(* CODESYS project Base_Elements.library
   Company: Vistaprint
   Title: Base_Elements
   Description: 0.0.1.22 - FB_UMC Always SingleAnswer 
      0.0.1.21 - Added GHT (10Digit Key compatible Hash)
      0.0.1.20 - Added newest BasePLC, addapted main component controll
      0.0.1.19 - Added newest EtherCat Library version
      0.0.1.18 - FB_BCC RP-208 - Implement sensor signal input for triggering a barcode scan
      0.0.1.17 - DRV Main Switch added
      0.0.1.16 - Added the Generic DataChannels
      0.0.1.15 - Added new BaseConcept Lib V0.3.4.8
      0.0.1.14 - Added new BaseConcept Lib
      0.0.1.13 - Changes in timeout handling BaseCtrlModule. Inserted new parameter  udiTimeoutStarting_ms. TO handling can now switched off with value 0.
      0.0.1.12 - Added new base_class
      0.0.1.11 - Bugfix in UMC
      0.0.1.10 - SGT added
      0.0.1.9 - Newest Base_PLC added 0.3.4.5
      0.0.1.8 - Integrate ECD (EtherCAT Diagnostic)
      0.0.1.7 - More RFW Error information
      0.0.1.5 - Added new controller FB_VLV
      0.0.1.4 - Fix for the BCD, BCC controller to support also messages without diagnostics
      0.0.1.2 - Simulation UMC; FB_CtrlModule added
      0.0.1.1 - Newest Base_PLC added 0.3.4.2
      0.0.1.0 - Newest Base_PLC added 0.3.4.0
      - FB_RFW Bug fix write single data
      0.0.0.26 - FB_ACL Enter ADS route string automatically during state PONBusy.
      0.0.0.25 - DLL FUB added
      0.0.0.24 - EOFFbusy Fix in FB_UMC
      0.0.0.23 - New ADS Client FUB (ACL) added
      	Sample added in MiddleTask
      0.0.0.22 - UMC simulation added, Refactoring
      0.0.0.21 - UMC - Add EMO State, Refactoring
      0.0.0.20 - New version of BCD and BCC
      0.0.0.19 - Back to BasePLC Lib. V3.3.5 beacuase of PageFaults
      0.0.0.18 - RFW integrated from Promp
      0.0.0.17 - DRV added
      0.0.0.16 - Newest Base_PLC added 0.3.3.7
      0.0.0.15 - Basic versions of Barcode driver and controller added
      0.0.0.11 - Newest Base_PLC added
      0.0.0.10 - Newest Base_PLC added
      0.0.0.9 - Add cylinder Level0, Update to Base PLC 0.3.3.2
      0.0.0.8 - Update to Base PLC 0.3.3.0
      0.0.0.7 - Updated to newest tc2_utilities
      0.0.0.6 - Added the PRS controller
      0.0.0.5 - Added the UMC and VPC controller
   Author: DSC - KVO
   Version: 0.0.1.22

Project tree, tasks and I/O mapping:
  libraries: Base_PLC, 0.3.4.9 (Vistaprint); Tc2_EtherCAT, 3.3.3.0 (Beckhoff Automation GmbH); Tc2_SerialCom, 3.3.2.0 (Beckhoff Automation GmbH); Tc2_Standard, 3.3.0.0 (Beckhoff Automation GmbH); Tc2_System, 3.3.5.0 (Beckhoff Automation GmbH); Tc2_TcpIp, 3.3.2.0 (Beckhoff Automation GmbH); Tc2_Utilities, 3.3.7.0 (Beckhoff Automation GmbH); Tc3_Interfaces, 3.3.0.0 (Beckhoff Automation GmbH); Tc3_MemMan, 3.3.1.0 (Beckhoff Automation GmbH); Tc3_Module, 3.3.5.0 (Beckhoff Automation GmbH)
  POUs/
    Controller/
      Driver/
        ACL (ADS client for data exchange)/
          global variables ACL_Const
          global variables ADS_IndexGroup
          data type E_ADS_AccessType
          function block FB_ACL [ST]: AddConnection, Always, FB_init, getCmdState, getCtrlSIf, GetNextAccessType, NetIDtoAddress, sta_ERROR, sta_OFF, sta_PON, sta_PONBusy, sta_RUN, sta_RUNBusy, StateMachine
          data type T_ADS_ConnectionData
          data type T_Ctrl_SIf_ACL
          data type T_Ctrl_SIf_ACL_Cur
          data type T_Ctrl_SIf_ACL_Par
        BCD (Bar code driver)/
          global variables BCD_CmdState
          function block FB_BCD [ST]: CheckSensorError, CtrlInit, CycleEndDuty, CycleStartDuty, FB_init, getCmdState, getSIf, HandleRxData, HandleTxData, PrepareBarCodeData, PrepareReadMsg, PrepareSendMsg, sta_CloseSocketBusy, sta_ComTestBusy, sta_ConnectSocketBusy, sta_Error, sta_ReadCodeBusy, sta_SocketClosed, sta_WaitForJob, StateMachine
          function FC_StrComp [ST]
          data type T_BCD
          data type T_BCD_Cfg
          data type T_BCD_Data
          data type T_BCD_DeviceInfo
          data type T_BCD_Error
          data type T_BCD_OperatingData
          data type T_BCD_Par
          data type T_BCD_ServiceInfo
          data type T_BCD_StateMachine
          data type T_BCD_Status
        PRS [Present Sensor]/
          data type E_ALM_PRS
          function block FB_PRS [ST]: Always, CtrlSIf, FB_init, getCmdState, getCtrlSIf, IoInBridge, IoOutBridge, sta_ABSENT, sta_ABSENTBusy, sta_PON, sta_PRESENT, sta_PRESENTBusy, StateMachine
          global variables PRS_CmdState
          data type T_Ctrl_SIf_PRS
          data type T_Ctrl_SIf_PRS_Cfg
          data type T_Ctrl_SIf_PRS_Cur
          data type T_Ctrl_SIf_PRS_Ilk
          data type T_Ctrl_SIf_PRS_In
          data type T_Ctrl_SIf_PRS_Out
          data type T_Ctrl_SIf_PRS_Par
        RFD (RFID Driver)/
          data type E_Typ_Baudrate
          data type E_Typ_Ftim
          function block FB_Com_3964R [ST]
          function block FB_ExCom [ST]
          function FB_HEXSTRING_TO_ULINT [ST]
          function block FB_RFD [ST]: CtrlInit, CycleEndDuty, CycleStartDuty, FB_init, getCmdState, getSIf, sta_CheckBusy, sta_Error, sta_MDSBusy, sta_Off, sta_OffBusy, sta_PowerOnBusy, sta_ReadBusy, sta_SLGBusy, sta_TagInitBusy, sta_WaitForJob, sta_WriteBusy, StateMachine, StateMachine_Service
          function block FB_RFR [ST]: CtrlInit, CycleEndDuty, CycleStartDuty, FB_init, getCmdState, getSIf, sta_Error, sta_PowerOnBusy, sta_WaitForJob, StateMachine, StateMachine_Service
          global variables RFD_Cmd
          global variables RFD_Constants
          data type T_RFD
          data type T_RFD_Cfg
          data type T_RFD_Cur
          data type T_RFD_Error
          data type T_RFD_MDS_Diagnose
          data type T_RFD_MDS_State
          data type T_RFD_SLG_Diagnose
          data type T_RFD_SLG_State
          data type T_RFD_StateMachine
          data type T_RFD_Status
          data type T_StateWord
      Lvl0/
        BCC (Barcode controller)/
          global variables BCC_CmdState
          function block FB_BCC [ST]: Always, FB_init, getCmdState, getCtrlSIf, IoInBridge, IoOutBridge, sta_ERROR, sta_OFF, sta_OFFBusy, sta_PON, sta_PONBusy, sta_READ, sta_READBusy, StateMachine
          data type T_BCC_Data
          data type T_Ctrl_SIf_BCC
          data type T_Ctrl_SIf_BCC_Cfg
          data type T_Ctrl_SIf_BCC_Cur
          data type T_Ctrl_SIf_BCC_In
          data type T_Ctrl_SIf_BCC_Out
          data type T_Ctrl_SIf_BCC_Par
        CYL (Cylinder)/
          global variables CYL_CmdState
          data type E_ALM_CYL
          data type E_Typ_CYL
          function block FB_CYL [ST]: Always, FB_init, getCmdState, getCtrlSIf, IoInBridge, IoOutBridge, sta_ERROR, sta_ERRORQuit, sta_EXTEND, sta_EXTENDBusy, sta_OFF, sta_OFFBusy, sta_RETRACT, sta_RETRACTBusy, sta_STOP, sta_STOPBusy, StateMachine
          data type T_Ctrl_SIf_CYL
          data type T_Ctrl_SIf_CYL_Cfg
          data type T_Ctrl_SIf_CYL_Cur
          data type T_Ctrl_SIf_CYL_Ilk
          data type T_Ctrl_SIf_CYL_In
          data type T_Ctrl_SIf_CYL_Out
          data type T_Ctrl_SIf_CYL_Par
        DRV (Drive)/
          global variables Const_DRV
          data type E_Typ_DRV
          function block FB_DRV [ST]: Always, FB_init, getCtrlSIf, IoInBridge, IoOutBridge, SetSpeed, sta_ERROR, sta_OFF, sta_OFFBusy, sta_PON, sta_RUN, sta_RUNBusy, StateMachine
          data type T_Ctrl_SIf_DRV
          data type T_Ctrl_SIf_DRV_Cfg
          data type T_Ctrl_SIf_DRV_Cur
          data type T_Ctrl_SIf_DRV_In
          data type T_Ctrl_SIf_DRV_Out
          data type T_Ctrl_SIf_DRV_Par
        ECD (EtherCAT Diagnostic)/
          data type E_ALM_ECD
          global variables ECD_Const
          function block FB_ECD [ST]: Always, FB_init, getCmdState, getCtrlSIf, sta_ERROR, sta_ERRORQuit, sta_OFF, sta_PON, sta_PONBusy, sta_RUN, sta_RUNBusy, StateMachine
          data type T_Ctrl_SIf_ECD
          data type T_Ctrl_SIf_ECD_Cfg
          data type T_Ctrl_SIf_ECD_Cur
          data type T_Ctrl_SIf_ECD_Par
          data type T_ECD_SlaveData
        RFW (RFID Reader-Writer)/
          data type E_Typ_RFW
          function block FB_DtChnToLine_NewRFID [ST]: Creat
          function block FB_RFW [ST]: Always, FB_init, getCmdState, getCtrlSIf, IoInBridge, IoOutBridge, sta_ERROR, sta_OFF, sta_OFFBusy, sta_ON, sta_ONbusy, sta_PON, sta_PONBusy, sta_READ, sta_READBusy, sta_RUN, sta_RUNbusy, sta_WRITE, sta_WRITEBusy, StateMachine
          function FB_ULINT_TO_HEXSTRING [ST]
          global variables RFID_Data
          global variables RFW_CmdState
          data type T_Ctrl_SIf_RFW
          data type T_Ctrl_SIf_RFW_Cfg
          data type T_Ctrl_SIf_RFW_Cur
          data type T_Ctrl_SIf_RFW_DtChnToLine
          data type T_Ctrl_SIf_RFW_In
          data type T_Ctrl_SIf_RFW_Out
          data type T_Ctrl_SIf_RFW_Par
          data type T_NewRFID_DtChn
          data type T_RFW
        SGT (Signal Tower)/
          data type E_ALM_SGT
          function block FB_SGT [ST]: Always, FB_init, getCmdState, getCtrlSIf, IoOutBridge, setBeepOutput, setLampOutput, sta_OFF, sta_OFFBusy, sta_PON, sta_PONBusy, sta_RUN, sta_RUNBusy, StateMachine
          data type T_Ctrl_SIf_SGT
          data type T_Ctrl_SIf_SGT_Cfg
          data type T_Ctrl_SIf_SGT_Out
          data type T_Ctrl_SIf_SGT_Par
        UMC [Universal Motor Controller]/
          data type E_ALM_UMC
          data type E_CFG_UMC
          data type E_TURN_DIRECTION
          data type E_UMC_MOTOR_STATUS
          function block FB_UMC [ST]: Always, cmd_MotorOff, cmd_MotorOn, cmd_MotorReset, cmd_MotorStop, CtrlInit, CtrlSIf, CycleEndDuty, CycleStartDuty, FB_init, getCmdState, getCtrlSIf, GetMotorStatus, GetSpeedValue, IoInBridge, IoOutBridge, sta_EOFF, sta_EOFFbusy, sta_ERROR, sta_ERRORQuit, sta_OFF, sta_OFFBusy, sta_PON, sta_RESETMOTORERROR, sta_RUN, sta_RUNBusy, sta_SETOPERATIONMODE, sta_STOP, sta_STOPBusy, StateMachine
          data type T_Ctrl_SIf_UMC
          data type T_Ctrl_SIf_UMC_Cfg
          data type T_Ctrl_SIf_UMC_Cur
          data type T_Ctrl_SIf_UMC_Ilk
          data type T_Ctrl_SIf_UMC_In
          data type T_Ctrl_SIf_UMC_Out
          data type T_Ctrl_SIf_UMC_Par
          data type T_UMC_Lenze_Control
          data type T_UMC_Lenze_Status
          data type U_UMC_Lenze_Control
          data type U_UMC_Lenze_Status
          global variables UMC_CmdState
        VLV (Valve controller)/
          data type E_ALM_VLV
          data type E_Typ_VLV
          function block FB_VLV [ST]: Always, FB_init, getCmdState, getCtrlSIf, IoInBridge, IoOutBridge, sta_CLOSE, sta_CLOSEBusy, sta_ERROR, sta_ERRORQuit, sta_OFF, sta_OFFBusy, sta_OPEN, sta_OPENBusy, StateMachine
          data type T_Ctrl_SIf_VLV
          data type T_Ctrl_SIf_VLV_Cfg
          data type T_Ctrl_SIf_VLV_Cur
          data type T_Ctrl_SIf_VLV_Ilk
          data type T_Ctrl_SIf_VLV_In
          data type T_Ctrl_SIf_VLV_Out
          data type T_Ctrl_SIf_VLV_Par
          global variables VLV_CmdState
        VPC [Vacuum Pump Controller]/
          data type E_ALM_VPC
          data type E_CFG_VPC
          function block FB_VPC [ST]: Always, FB_init, getCmdState, getCtrlSIf, IoInBridge, IoOutBridge, sta_ERROR, sta_ERRORQuit, sta_OFF, sta_OFFBusy, sta_PON, sta_RUN, sta_RUNBusy, sta_StabilizeVacuum, StateMachine
          data type T_Ctrl_SIf_VPC
          data type T_Ctrl_SIf_VPC_Cfg
          data type T_Ctrl_SIf_VPC_Cur
          data type T_Ctrl_SIf_VPC_Ilk
          data type T_Ctrl_SIf_VPC_In
          data type T_Ctrl_SIf_VPC_Out
          data type T_Ctrl_SIf_VPC_Par
          global variables VPC_CmdState
      Lvl1/
      Lvl2/
      Lvl3/
        BaseCtrlModule/
          function block FB_CtrlModule [ST]: AddIBufferChilds, AddIBufferFullChilds, AddSeqChild, Always, checkChildAlmClass, checkValidPointer, CtrlInit, FB_init, getCmdState, IoInBridge, IoOutBridge, SIf_Cfg, SIf_Cur, SIf_In, SIf_Par, sta_EOFF, sta_EOFFBusy, sta_ERROR, sta_OFF, sta_RUN, sta_RUNBusy, sta_STOP, sta_STOPBusy, StateMachine
          function block FB_IBuffer [ST]: BufferFull, MaxCapacity, NumOfHangers
          interface IBuffer: BufferFull, MaxCapacity, NumOfHangers
          data type T_Ctrl_SIf_MOD
          data type T_Ctrl_SIf_MOD_Cfg
          data type T_Ctrl_SIf_MOD_Cur
          data type T_Ctrl_SIf_MOD_In
          data type T_Ctrl_SIf_MOD_Par
          data type T_Sequence
    Utility/
      AFF [Array Fifo]/
        function block FB_ArrayFifo [ST]: FreePointer, Initialize, ItemCount, MaxBufferSize, Peek, Pop, Push, Reset
      Data Channel/
        IdBase/
          function block FB_IdBaseRecvDch [ST]: GetData, InitChannel
          function block FB_IdBaseSendDch [ST]: InitChannel, SendData
          global variables IdBaseConst
          data type T_IdBaseRecvData
          data type T_IdBaseSendData
      DCH [Data Channel Base]/
        data type E_DCH_Error
        data type E_PlcSaberDHCState
        data type E_SaberPlcDHCState
        function block FB_DataChannelRecvBase [ST]: Busy, DataSize, Error, GetData, InitChannel
        function block FB_DataChannelRecvFifo [ST]: DataChannel, Enable, Item, MaxFifoSize
        function block FB_DataChannelSendBase [ST]: Busy, DataSize, Error, InitChannel, SendData
        function block FB_DataChannelSenderFifo [ST]: DataChannel, Enable, MaxFifoSize
        interface I_DataChannelRecv: Busy, DataSize, Error, GetData, InitChannel
        interface I_DataChannelSend: Busy, DataSize, Error, InitChannel, SendData
      DFF [Dynamic Pointer FiFo]/
        function block FB_DynamicFifo [ST]: ClearFifo, FreeDataPointer, ItemCount, Peek, Pop, Push
      GHT [Generic Hash Table]/
        function block FB_GHT [ST]: AddItem, Clear, Count, FB_init, GetTableIdx, Initialize, Lookup
        interface IGHT: AddItem, Clear, Count, Initialize, Lookup
        data type T_GHTHashTableBuffer
      ItemBase/
        data type E_Destination
        data type E_ItemHealth
        data type E_PrintSelection
        global variables ItemConst
        data type T_IdBase_DCH
        data type T_ItemBase
        data type T_ItemPaperBase
        data type T_QueueBase
  Version/
    global variables Global_Version
*)

// POUs/Controller/Driver/ACL (ADS client for data exchange)/E_ADS_AccessType
TYPE E_ADS_AccessType :
(
	READ := 0,
	WRITE := 1
);
END_TYPE

// POUs/Controller/Driver/ACL (ADS client for data exchange)/T_ADS_ConnectionData
TYPE T_ADS_ConnectionData :
STRUCT
	// Connection ID. Automatically assigned by calling method for adding new connection
	udiConID: UDINT;
	// Handle ID for data exchange. Determined automatically during state PONbusy.
	udiHandle: UDINT;
	// Route of the PRG or FUB instance on server side. Example: 'SlowPRG_1.fbData.SIf.cur.st_ADSData'
	strRoute: STRING;
	// ADS target port
	uinTargetPort: UINT;
	/// NetID
	strNetID: STRING(30);
	// Access type
	eAccessType: E_ADS_AccessType;
	// Length of the data structure
	udiDataLen: UDINT;
	// Pointer to data structure. Note: Defined structure must be the same on client and server side.
	pData: PVOID;
END_STRUCT
END_TYPE

// POUs/Controller/Driver/ACL (ADS client for data exchange)/T_Ctrl_SIf_ACL
TYPE T_Ctrl_SIf_ACL :
STRUCT
	// parameter
	Par: T_Ctrl_SIf_ACL_Par;
	// current values
	Cur: T_Ctrl_SIf_ACL_Cur;
	// alarm number used in this controller
	Alm: ARRAY[1..7] OF T_Ctrl_Alm;
END_STRUCT
END_TYPE

// POUs/Controller/Driver/ACL (ADS client for data exchange)/T_Ctrl_SIf_ACL_Cur
TYPE T_Ctrl_SIf_ACL_Cur :
STRUCT
	// Shows the number of ADS (server) connections
	uinNumOfAdsConnections: UINT;
END_STRUCT
END_TYPE

// POUs/Controller/Driver/ACL (ADS client for data exchange)/T_Ctrl_SIf_ACL_Par
TYPE T_Ctrl_SIf_ACL_Par :
STRUCT
	// [ms] Timeout power on. Timeout for initialize all ADS connections.
	udiTOPowerOn_ms: UDINT;
	// [ms] Timeout add route
	udiTOAddRoute_ms: UDINT;
	// [ms] Timeout read data
	udiTOReadData_ms: UDINT;
	// [ms] Timeout write data
	udiTOWriteData_ms: UDINT;
	// [ms] Timeout read/write data
	udiTORWData_ms: UDINT;
	// [ms] Polling interval for read/write of all ADS connections in list
	udiPollingInterval_ms: UDINT;
END_STRUCT
END_TYPE

// POUs/Controller/Driver/BCD (Bar code driver)/T_BCD
TYPE T_BCD :
STRUCT
	strState: STRING;
	strCmd: STRING;
	intCmd: INT;
	stStatus: T_BCD_Status;
	stErr: T_BCD_Error;
	stCfg: T_BCD_Cfg;
	stPar: T_BCD_Par;
	stData: T_BCD_Data;
END_STRUCT
END_TYPE

// POUs/Controller/Driver/BCD (Bar code driver)/T_BCD_Cfg
TYPE T_BCD_Cfg :
STRUCT
	bolSimulation: BOOL;
	strSensorIPAdr: STRING(15) := '';
	udiSensorPort: UDINT := 0;
	/// Barcode is also sending diagnostics data
	bolResponseIncludingDiagnostics			: BOOL;
END_STRUCT
END_TYPE

// POUs/Controller/Driver/BCD (Bar code driver)/T_BCD_Data
TYPE T_BCD_Data :
STRUCT
	bolCodeReaded: BOOL;
	uliBarCode: ULINT;
	strBarCode: STRING;
	stDevInfo: T_BCD_DeviceInfo;
	stServInfo: T_BCD_ServiceInfo;
	stOpData: T_BCD_OperatingData;
END_STRUCT
END_TYPE

// POUs/Controller/Driver/BCD (Bar code driver)/T_BCD_DeviceInfo
TYPE T_BCD_DeviceInfo :
STRUCT
	strComTestResult: STRING(40);
	strManufacturer: STRING(25);
	strDeviceType: STRING(25);
	strOrderNumber: STRING(20);
	strSWVersion: STRING(10);
	/// shows the firmware version of the device
	strFWVersion: STRING(10);
	strSerialNumber: STRING(20);
END_STRUCT
END_TYPE

// POUs/Controller/Driver/BCD (Bar code driver)/T_BCD_Error
TYPE T_BCD_Error :
STRUCT
	/// Reset failure
	bolErrAck: BOOL;
	/// atleast one failure active
	bolErrorActive: BOOL;
	/// error in TCP socket
	bolSocketError: BOOL;
	/// error in sensor (SICK)
	bolSensorError: BOOL;
	/// error ID
	udiErrorID: UDINT;
END_STRUCT
END_TYPE

// POUs/Controller/Driver/BCD (Bar code driver)/T_BCD_OperatingData
TYPE T_BCD_OperatingData :
STRUCT
	strPowerOnCounter: STRING(25);
	strOpHours: STRING(25);
	strPowerOnHours: STRING(20);
END_STRUCT
END_TYPE

// POUs/Controller/Driver/BCD (Bar code driver)/T_BCD_Par
TYPE T_BCD_Par :
STRUCT
	tTOConnection: TIME;
	tTOSend: TIME;
	tTOReceive: TIME;
END_STRUCT
END_TYPE

// POUs/Controller/Driver/BCD (Bar code driver)/T_BCD_ServiceInfo
TYPE T_BCD_ServiceInfo :
STRUCT
	strLastUsername: STRING(25);
	strLastParChangeDate: STRING(10);
	strLastParChangeTime: STRING(5);
END_STRUCT
END_TYPE

// POUs/Controller/Driver/BCD (Bar code driver)/T_BCD_StateMachine
TYPE T_BCD_StateMachine :
STRUCT
	/// actual state
	intState: INT;
	/// state of last cycle
	intStateLastCycle: INT;
	/// save history backup p.e. in ERROR state
	intStateHistory: INT;
	/// set state for next cycle
	intStateNext: INT;
	/// Time in this State
	udiTimeInState_ms: UDINT;
END_STRUCT
END_TYPE

// POUs/Controller/Driver/BCD (Bar code driver)/T_BCD_Status
TYPE T_BCD_Status :
STRUCT
	/// Socket connected
	bolSocketConnected: BOOL;
	bolComChecked: BOOL;
END_STRUCT
END_TYPE

// POUs/Controller/Driver/PRS [Present Sensor]/E_ALM_PRS
TYPE E_ALM_PRS :
(
	Dummy		 		:= 1,
	MAX_E_ALM_PRS
) UINT;
END_TYPE

// POUs/Controller/Driver/PRS [Present Sensor]/T_Ctrl_SIf_PRS
TYPE T_Ctrl_SIf_PRS :
STRUCT
	///configuration
	Cfg: T_Ctrl_SIf_PRS_Cfg;
	///parameter
	Par: T_Ctrl_SIf_PRS_Par;
	///current values
	Cur: T_Ctrl_SIf_PRS_Cur;
	///io input
	In: T_Ctrl_SIf_PRS_In;
	///io output
	Out: T_Ctrl_SIf_PRS_Out;
	///alarm number used in this controller
	Alm: ARRAY[1..E_ALM_PRS.MAX_E_ALM_PRS] OF T_Ctrl_Alm;
	///interlock of output/movements
	Ilk: T_Ctrl_SIf_PRS_Ilk;
END_STRUCT
END_TYPE

// POUs/Controller/Driver/PRS [Present Sensor]/T_Ctrl_SIf_PRS_Cfg
TYPE T_Ctrl_SIf_PRS_Cfg :
STRUCT
END_STRUCT
END_TYPE

// POUs/Controller/Driver/PRS [Present Sensor]/T_Ctrl_SIf_PRS_Cur
TYPE T_Ctrl_SIf_PRS_Cur :
STRUCT	
END_STRUCT
END_TYPE

// POUs/Controller/Driver/PRS [Present Sensor]/T_Ctrl_SIf_PRS_Ilk
TYPE T_Ctrl_SIf_PRS_Ilk :
STRUCT
END_STRUCT
END_TYPE

// POUs/Controller/Driver/PRS [Present Sensor]/T_Ctrl_SIf_PRS_In
TYPE T_Ctrl_SIf_PRS_In :
STRUCT
	/// Input Sensor is present
	bolPresent					: BASE_PLC.T_Ctrl_IoBool;
END_STRUCT
END_TYPE

// POUs/Controller/Driver/PRS [Present Sensor]/T_Ctrl_SIf_PRS_Out
TYPE T_Ctrl_SIf_PRS_Out :
STRUCT
END_STRUCT
END_TYPE

// POUs/Controller/Driver/PRS [Present Sensor]/T_Ctrl_SIf_PRS_Par
TYPE T_Ctrl_SIf_PRS_Par :
STRUCT
	/// [ms] Debounce time until it shows as present
	udiDebouncePresentTime_ms				: UDINT;
	/// [ms] Debounce time until it shows as absent
	udiDebounceAbsentTime_ms	    		: UDINT;
	/// True = simulated hanger available
	bolSimHangerAvailable					: BOOL;
END_STRUCT
END_TYPE

// POUs/Controller/Driver/RFD (RFID Driver)/E_Typ_Baudrate
TYPE E_Typ_Baudrate :
(
	baud_2400 := 4,
	baud_4800 := 5,
	baud_9600 := 6,
	baud_19200 := 7,
	baud_38400 := 8,
	baud_57600 := 9,
	baud_115200 := 10
);
END_TYPE

// POUs/Controller/Driver/RFD (RFID Driver)/E_Typ_Ftim
TYPE E_Typ_Ftim :
(
	/// Setting for air interface
	RF300 := 0,
	ISO_generall := 1,
	ISO_infineon := 3,
	ISO_Fujitsu := 4,
	ISO_NXP := 5,
	ISO_TI := 6,
	ISO_ST := 7,
	Max_E_Typ_Ftim
);
END_TYPE

// POUs/Controller/Driver/RFD (RFID Driver)/T_RFD
TYPE T_RFD :
STRUCT
	strState: STRING;
	strCmd: STRING;
	intCmd: INT;
	intServiceCmd: INT;
	stStatus: T_RFD_Status;
	stCfg: T_RFD_Cfg;
	stCur: T_RFD_Cur;
	stErr: T_RFD_Error;
END_STRUCT
END_TYPE

// POUs/Controller/Driver/RFD (RFID Driver)/T_RFD_Cfg
TYPE T_RFD_Cfg :
STRUCT
	bolSimulation: BOOL;
	eTyp: E_Typ_RFW;
	/// Reset parameter value
	usiResetParameter: USINT := 2#101010;
	/// Setting of the Air interface
	usiFtimSetting: E_Typ_Ftim;
	/// Reset option1 value
	usiResetOption1: USINT := 2#10;
	/// Set Baudrate
	uinBaudrate: USINT;
	/// Set Communikationsettings
	uinComSettings: USINT;
	/// Net ID oft EtherCat Master
	stNetId: TC2_SYSTEM.T_AmsNetID;
	/// Port Number of EtherCat Slave Comunication Module
	uinSlaveAddr: UINT;
	/// CoE Object Index for Communication Settings
	uinCoeIndexComSettings: WORD := 16#8000;
	/// CoE Object SubIndex for Baudrate
	usiCoeSubindexComBaudrate: BYTE := 16#11;
	/// CoE Object SubIndex for Dataframe
	usiCoeSubindexComDataframe: BYTE := 16#15;
	/// Retry Job to RFID Reader
	udiRetry: UDINT := 10;
	//////////////////////////////////////////////////
	/// Reset Memory 00=RAM, 01=remanent
	usiMemory: USINT := 0;
	/// Scan Mode 00= Continous Read; 01=Single Read
	usiScanMode: USINT := 1;
	/// Lock Time in ms
	uinLockTime_ms: UINT := 5000;
END_STRUCT
END_TYPE

// POUs/Controller/Driver/RFD (RFID Driver)/T_RFD_Cur
TYPE T_RFD_Cur :
STRUCT
	/// Pointer to Received Data Array
	pData: POINTER TO ARRAY[0..255] OF BYTE;
	/// Startadress to Read/Write at the data Array Element
	uinAdressData: UINT;
	/// Startadress to Read/Write at the Tag
	uinAdressTag: UINT;
	/// Number of bytes to Read/Write
	usiCount: USINT;
END_STRUCT
END_TYPE

// POUs/Controller/Driver/RFD (RFID Driver)/T_RFD_Error
TYPE T_RFD_Error :
STRUCT
	/// Reset failure
	bolErrAck: BOOL;
	/// atleast one failure active
	bolErrorActive: BOOL;
	/// error at communication card
	bolComError: BOOL;
	bolProtcolError: BOOL;
	/// Error with RF ID Tag
	bolRFIDError: BOOL;
	/// Error at setting of the communication Card (SDO Write)
	bolSDOError: BOOL;
	/// information to Communication Card error
	udiErrorID: UDINT;
END_STRUCT
END_TYPE

// POUs/Controller/Driver/RFD (RFID Driver)/T_RFD_MDS_Diagnose
TYPE T_RFD_MDS_Diagnose :
STRUCT
	/// Power flux density: as smaller the value, as higher the field intensity
	usiLFD: USINT;
	/// Errorcounter inactive mode
	usiFZP: USINT;
	/// Errorcounter active: CRC or signature errors
	usiFZA: USINT;
	/// Presence time of tag, resolution in 9.7ms
	usiANWZ: USINT;
END_STRUCT
END_TYPE

// POUs/Controller/Driver/RFD (RFID Driver)/T_RFD_MDS_State
TYPE T_RFD_MDS_State :
STRUCT
	/// MDS Type 1=no FRAM; 2=8k FRAM; 3=32k FRAM; 4=64k FRAM; 5=128k FRAM; 6=256k FRAM
	bytMDSType: BYTE;
	/// Lock bit registers (lock state)
	bytLockState: BYTE;
	/// MDS Version
	bytVersion: BYTE;
	/// Memory Size
	worMemSize: WORD;
	/// Blocksize in Byte
	bytBlockSize: BYTE;
	/// Value of memory Blocks
	bytBlockNo: BYTE;
END_STRUCT
END_TYPE

// POUs/Controller/Driver/RFD (RFID Driver)/T_RFD_SLG_Diagnose
TYPE T_RFD_SLG_Diagnose :
STRUCT
	/// Mode SLG Diagnose
	usiS_Info: USINT;
	/// Errorcounter inactive mode
	usiFZP: USINT;
	/// Counter abort
	usiABZ: USINT;
	/// Errorcounter code errors
	usiCFZ: USINT;
	/// Errorcounter signature errors
	usiSFZ: USINT;
	/// Errorcounter CRC
	usiCRCFZ: USINT;
	/// Actual command state
	usiBSTAT: USINT;
	/// Counter interface errors to host (Parity, BCC, Frame)
	usiASMFZ: USINT;
END_STRUCT
END_TYPE

// POUs/Controller/Driver/RFD (RFID Driver)/T_RFD_SLG_State
TYPE T_RFD_SLG_State :
STRUCT
	/// HW Type of SLG  0=RF310R RF340R RF350R (-xAA10); 1=RF380R (-3AA10); 2=RF310R(-1AB10); 3=RF380R (-3AB10); 4=RF340R RF350R (-2AB10,-4AB10)
	bytHWType: BYTE;
	/// HW Version
	worHWVersion: WORD;
	/// Loading Version
	worURLVersion: WORD;
	/// FW Type
	bytFWType: BYTE;
	/// FW Version
	worFWVersion: WORD;
	/// Driver Type 1=3964R
	bytDriverType: BYTE;
	/// Driver Version
	worDriverVersion: WORD;
	/// Communication port 1=RS422, 2=RS232
	bytComm: BYTE;
	/// Communication Baud rate 1=19.2kBaud; 3=57.6kBaud; 5=115.2kBaud
	bytBaud: BYTE;
	/// sending power (only RF380R) 0=standard; 2=0.5W; 3=0.75W; 4=1W; 5=1.25W (default); 6=1.5W; 7=1.75W; 8=2W
	bytPower: BYTE;
	/// Number of maximal tags in the field
	bytMtag: BYTE;
	/// air interface 0=RF300; 1=ISO generall; 3=ISO infineon Chip; 4=ISO Fujitsu; 5=ISO NXP; 6=ISO TI; 7=ISO ST
	bytFtim: BYTE;
	/// State antenna 1=ON; 2=OFF
	bytAntenna: BYTE;
	/// Tag presence 0=No presence; 1=prexence
	bytPresence: BYTE;
END_STRUCT
END_TYPE

// POUs/Controller/Driver/RFD (RFID Driver)/T_RFD_StateMachine
TYPE T_RFD_StateMachine :
STRUCT
	///actual state
	intState: INT;
	///state of last cycle
	intStateLastCycle: INT;
	///save history backup p.e. in ERROR state
	intStateHistory: INT;
	///set state for next cycle
	intStateNext: INT;
	///Time in this State
	udiTimeInState_ms: UDINT;
END_STRUCT
END_TYPE

// POUs/Controller/Driver/RFD (RFID Driver)/T_RFD_Status
TYPE T_RFD_Status :
STRUCT
	/// 1 = Antenna is initialized  
	bolStartupOk: BOOL;
	/// 1 = Antenna is initialized  
	bolInitOk: BOOL;
	/// 1 = Antenna is on 
	bolOn: BOOL;
	/// 1 = tag is present  
	bolPresent: BOOL;
	/// 1 = Communication to SLG is OK  
	bolL_UEB: BOOL;
	/// SLG State only actual on demand 
	stSLG_State: T_RFD_SLG_State;
	/// SLG Diagnose only actual on demand 
	stSLG_Diag: T_RFD_SLG_Diagnose;
	/// SLG State only actual on demand  
	stMDS_State: T_RFD_MDS_State;
	/// SLG Diagnose only actual on demand  
	stMDS_Diag: T_RFD_MDS_Diagnose;
	/// Tag ID
	abyteUID: ARRAY[0..7] OF BYTE;
END_STRUCT
END_TYPE

// POUs/Controller/Driver/RFD (RFID Driver)/T_StateWord
TYPE T_StateWord :
STRUCT
	///Acknowledge the datachange of this Command bit
	bolTransmitAccepted: BOOL;
	///New Datat at the input
	bolReceiveRequest: BOOL;
	///0=Ready for Data exchange; 1=initialisation of the clam
	bolInputAccepted: BOOL;
	///Input Buffer is full, all new arriveing data lost
	bolBufferFull: BOOL;
	///Parity Error occured
	bolParityErr: BOOL;
	///Framing Error occured
	bolFramingErr: BOOL;
	///Overrun Error occured
	bolOverrunErr: BOOL;
	///Amounth of the reached Input Bytes
	usiInLenght: USINT;
END_STRUCT
END_TYPE

// POUs/Controller/Lvl0/BCC (Barcode controller)/T_BCC_Data
TYPE T_BCC_Data :
STRUCT
	uliBarCode: ULINT;
	strBarCode: STRING;
END_STRUCT
END_TYPE

// POUs/Controller/Lvl0/BCC (Barcode controller)/T_Ctrl_SIf_BCC
TYPE T_Ctrl_SIf_BCC :
STRUCT
	/// configuration
	Cfg: T_Ctrl_SIf_BCC_Cfg;
	/// parameter
	Par: T_Ctrl_SIf_BCC_Par;
	/// current values
	Cur: T_Ctrl_SIf_BCC_Cur;
	/// io input
	In: T_Ctrl_SIf_BCC_In;
	/// io output
	Out: T_Ctrl_SIf_BCC_Out;
	/// alarm number used in this controller
	Alm: ARRAY[1..6] OF T_Ctrl_Alm;
END_STRUCT
END_TYPE

// POUs/Controller/Lvl0/BCC (Barcode controller)/T_Ctrl_SIf_BCC_Cfg
TYPE T_Ctrl_SIf_BCC_Cfg :
STRUCT
	/// IP Adress of the sensor (PLC = Client, Sensor = Server)
	strSensorIPAdr: STRING(15) := '';
	/// Port number of the sensor
	udiSensorPort: UDINT := 0;
END_STRUCT
END_TYPE

// POUs/Controller/Lvl0/BCC (Barcode controller)/T_Ctrl_SIf_BCC_Cur
TYPE T_Ctrl_SIf_BCC_Cur :
STRUCT
	/// Sensor connected
	bolConnected: BOOL;
	/// Communication checked during PON
	bolComChecked: BOOL;
	/// 1 = new bar code readed 
	bolNewCodeReaded: BOOL;
	/// 1 = no code readed, answer *No Read* 
	bolNoRead: BOOL;
	/// Sensor data
	stData: T_BCC_Data;
END_STRUCT
END_TYPE

// POUs/Controller/Lvl0/BCC (Barcode controller)/T_Ctrl_SIf_BCC_In
TYPE T_Ctrl_SIf_BCC_In :
STRUCT
	// Sensor input for triggering a new barcode scan 
	bolSensorTrigScan: BASE_PLC.T_Ctrl_IoBool;
END_STRUCT
END_TYPE

// POUs/Controller/Lvl0/BCC (Barcode controller)/T_Ctrl_SIf_BCC_Out
TYPE T_Ctrl_SIf_BCC_Out :
STRUCT
END_STRUCT
END_TYPE

// POUs/Controller/Lvl0/BCC (Barcode controller)/T_Ctrl_SIf_BCC_Par
TYPE T_Ctrl_SIf_BCC_Par :
STRUCT
	/// [ms] Timeout power on
	udiTOPowerOn_ms: UDINT;
	/// [ms] Timeout read
	udiTORead_ms: UDINT;
	// [ms] Barcode scan delay time - Delay before a barcode scan will be triggered after a new product has been detected by trigger sensor input
	udiExecuteScanDelayTime_ms: UDINT;
END_STRUCT
END_TYPE

// POUs/Controller/Lvl0/CYL (Cylinder)/E_ALM_CYL
{attribute 'qualified_only' := ''}
TYPE E_ALM_CYL :
(
	SensorRetractAlwaysOn	:= 1,
	SensorExtendNotReached	:= 2,
	SensorExtendAlwaysOn	:= 3,
	SensorRetractNotReached	:= 4,
	InterlockExtend	:= 5,
	InterlockRetract := 6,	
	MAX_E_ALM
) UINT;
END_TYPE

// POUs/Controller/Lvl0/CYL (Cylinder)/E_Typ_CYL
TYPE E_Typ_CYL :
(
	///bistabile and two feedback sensors
	Valve2_Sensor2 := 0,
	///bistabile and extended feedback sensors	
	Valve2_SensorExtended,
	///bistabile and retracted feedback sensors	
	Valve2_SensorRetracted,
	///bistabile and no feedback sensors
	Valve2_Sensor0,
	///monostabile and 2 feedback sensors	
	Valve1_Sensor2,
	///monostabile and extended feedback sensors	
	Valve1_SensorExtended,
	///monostabile and retracted feedback sensor
	Valve1_SensorRetracted,
	///monostabile and no feedback sensors
	Valve1_Sensor0,
	Max_E_Typ_CYL
);
END_TYPE

// POUs/Controller/Lvl0/CYL (Cylinder)/T_Ctrl_SIf_CYL
TYPE T_Ctrl_SIf_CYL :
STRUCT
	///configuration
	Cfg: T_Ctrl_SIf_CYL_Cfg;
	///parameter
	Par: T_Ctrl_SIf_CYL_Par;
	///current values
	Cur: T_Ctrl_SIf_CYL_Cur;
	///io input
	In: T_Ctrl_SIf_CYL_In;
	///io output
	Out: T_Ctrl_SIf_CYL_Out;
	///alarm number used in this controller
	Alm: ARRAY[1..(E_ALM_CYL.MAX_E_ALM-1)] OF T_Ctrl_Alm;
	///interlock of output/movements
	Ilk: T_Ctrl_SIf_CYL_Ilk;
END_STRUCT
END_TYPE

// POUs/Controller/Lvl0/CYL (Cylinder)/T_Ctrl_SIf_CYL_Cfg
TYPE T_Ctrl_SIf_CYL_Cfg :
STRUCT
	eTyp: E_Typ_CYL;
END_STRUCT
END_TYPE

// POUs/Controller/Lvl0/CYL (Cylinder)/T_Ctrl_SIf_CYL_Cur
TYPE T_Ctrl_SIf_CYL_Cur :
STRUCT
	///[ms] time last movement to retract
	udiMoveTimeRetract: UDINT;
	///[ms] time last movement to extend
	udiMoveTimeExtend: UDINT;
END_STRUCT
END_TYPE

// POUs/Controller/Lvl0/CYL (Cylinder)/T_Ctrl_SIf_CYL_Ilk
TYPE T_Ctrl_SIf_CYL_Ilk :
STRUCT
	///interlock retraction of cylinder
	bolRetract: BOOL;
	///interlock extend of cylinder
	bolExtend: BOOL;
END_STRUCT
END_TYPE

// POUs/Controller/Lvl0/CYL (Cylinder)/T_Ctrl_SIf_CYL_In
TYPE T_Ctrl_SIf_CYL_In :
STRUCT
	///sensor feedback position extended reached
	bolExtended: T_Ctrl_IoBool;
	///sensor feedback position retracted reached
	bolRetracted: T_Ctrl_IoBool;
END_STRUCT
END_TYPE

// POUs/Controller/Lvl0/CYL (Cylinder)/T_Ctrl_SIf_CYL_Out
TYPE T_Ctrl_SIf_CYL_Out :
STRUCT
	///switch valve retract
	bolRetract: T_Ctrl_IoBool;
	///switch valve extend
	bolExtend: T_Ctrl_IoBool;
END_STRUCT
END_TYPE

// POUs/Controller/Lvl0/CYL (Cylinder)/T_Ctrl_SIf_CYL_Par
TYPE T_Ctrl_SIf_CYL_Par :
STRUCT
	///[ms] until failure to long time for extend
	udiExtendTime_ms: UDINT;
	///[ms] until failure to long time for retract
	udiRetractTime_ms: UDINT;
	///[ms] simulation time for extend or /2 of timeout time?
	udiSimExtendTime_ms: UDINT;
	///[ms] simulation time for retract or /2 of timeout time?
	udiSimRetractTime_ms: UDINT;
END_STRUCT
END_TYPE

// POUs/Controller/Lvl0/DRV (Drive)/E_Typ_DRV
TYPE E_Typ_DRV :
(
	None := 0,
	TLP,
	TLK,
	TLKV,
	TLPsort,
	TLS,
	TLC,
	Max_E_Typ_JUN
);
END_TYPE

// POUs/Controller/Lvl0/DRV (Drive)/T_Ctrl_SIf_DRV
TYPE T_Ctrl_SIf_DRV :
STRUCT
	///configuration
	Cfg: T_Ctrl_SIf_DRV_Cfg;
	///parameter
	Par: T_Ctrl_SIf_DRV_Par;
	///current values
	Cur: T_Ctrl_SIf_DRV_Cur;
	///io input
	In: T_Ctrl_SIf_DRV_In;
	///io output
	Out: T_Ctrl_SIf_DRV_Out;
	///alarm number used in this controller
	Alm: ARRAY[1..5] OF T_Ctrl_Alm;
END_STRUCT
END_TYPE

// POUs/Controller/Lvl0/DRV (Drive)/T_Ctrl_SIf_DRV_Cfg
TYPE T_Ctrl_SIf_DRV_Cfg :
STRUCT
	/// Type of drive
	eTyp: E_Typ_DRV;
	/// Distance per pulse	
	dinDistPerPulse_um: DINT;
	/// Has Variable Speed	
	bolSpeedVariable: BOOL;
	/// Has Pulse signal for position and speed calculation
	bolPulseExist: BOOL;
	/// Number of blocked supervision inputs
	usiCountBlockedSupervis: USINT;
	/// [um] PinDistance
	dinPinDistance_um: DINT;
	/// Enable Maintenace Switch
	bolEnableMaintenaceSwitch: BOOL;
END_STRUCT
END_TYPE

// POUs/Controller/Lvl0/DRV (Drive)/T_Ctrl_SIf_DRV_Cur
TYPE T_Ctrl_SIf_DRV_Cur :
STRUCT
	dinPulseCounter: DINT;
	dinPos_um: DINT;
	dinSpeed_um_s: DINT;
END_STRUCT
END_TYPE

// POUs/Controller/Lvl0/DRV (Drive)/T_Ctrl_SIf_DRV_In
TYPE T_Ctrl_SIf_DRV_In :
STRUCT
	bolOverload: T_Ctrl_IoBool;
	bolPulse: T_Ctrl_IoBool;
	a_bolBlockedSupvervis: ARRAY[1..cMAX_BLOCKED_SUP] OF BASE_PLC.T_Ctrl_IoBool;
	/// DI of Maintenance Switch
	bolMaintenanceSwitch: T_Ctrl_IoBool;
END_STRUCT
END_TYPE

// POUs/Controller/Lvl0/DRV (Drive)/T_Ctrl_SIf_DRV_Out
TYPE T_Ctrl_SIf_DRV_Out :
STRUCT
	/// bolSpeed_1 = slow
	/// bolSpeed_2 = fast
	/// bolSpeed_1 & bolSpeed_2 = middle speed 
	bolSpeed_1: T_Ctrl_IoBool;
	bolSpeed_2: T_Ctrl_IoBool;
END_STRUCT
END_TYPE

// POUs/Controller/Lvl0/DRV (Drive)/T_Ctrl_SIf_DRV_Par
TYPE T_Ctrl_SIf_DRV_Par :
STRUCT
	/// [ms] Timeout supervision of pulse in RUN
	udi_pulseTimeout_ms: UDINT;
	/// [ms] Simulation of pulse in RUN: 0.676mm/ms / 38.4mm/puls => 56.8ms/puls
	udi_pulseSim_ms: UDINT;
	/// 0=slow, 1=middle, 2=fast
	usi_speedLevel: USINT;
	/// Maximum Broken Pins
	int_MaxBrokenPins: INT;
END_STRUCT
END_TYPE

// POUs/Controller/Lvl0/ECD (EtherCAT Diagnostic)/E_ALM_ECD
TYPE E_ALM_ECD :
(
	/// ADS Communication Error to EtherCAT Master => Info = ADS_Errorcode
	ADS_ComError := 1,
	/// A Function is not finished after the defined Timeout
	TimeOutFunction := 2,
	/// Configured and reached Slaves are not the same => Info Byte 0+1 = Slave Addres from last error Info Byte 2+3 = Numbers of error Slaves
	NotAllSlaveConnected := 3,
	/// More slaves at the master as the structure could handle => Info Byte 0+1 = Slave Addres from last error Info Byte 2+3 = Numbers of error Slaves
	ToManySlaves := 4,
	/// Master not in the correct state => Info = Masterstate
	MasterStateError := 5,
	/// Minimum one Slave not in the correct state => Byte 0+1 = Slave Addres from last error, Info Byte 2 + 3 = State of last error Slave
	SlaveStateError := 6,
	/// Minimum one Slave has to many CRC Erros => Byte 0+1 = Slave Addres from last error, Info Byte 2 +3 = Number of CRC Errors from last Slave with error
	SlaveCRCError := 7,
	/// Minimum one Slave has a LinkState Erros => Byte 0+1 = Slave Addres from last error Info Byte 2 + 3 = Link State of last error Slave
	SlaveLinkError := 8,
	/// No slave found in the network
	NoSlaveFound := 9,
	/// To many abnormal State Changes
	StateChanges := 10,
	MAX_E_ALM
) UINT;
END_TYPE

// POUs/Controller/Lvl0/ECD (EtherCAT Diagnostic)/T_Ctrl_SIf_ECD
TYPE T_Ctrl_SIf_ECD :
STRUCT
	/// configuration
	Cfg: T_Ctrl_SIf_ECD_Cfg;
	/// parameter
	Par: T_Ctrl_SIf_ECD_Par;
	/// current values
	Cur: T_Ctrl_SIf_ECD_Cur;
	/// alarm number used in this controller
	Alm: ARRAY[1..(E_ALM_ECD.MAX_E_ALM - 1)] OF T_Ctrl_Alm;
END_STRUCT
END_TYPE

// POUs/Controller/Lvl0/ECD (EtherCAT Diagnostic)/T_Ctrl_SIf_ECD_Cfg
TYPE T_Ctrl_SIf_ECD_Cfg :
STRUCT
	/// NetID
	strNetID: STRING(30);
	/// Run allways the scanning without set into run
	bolRunAlways: BOOL;
END_STRUCT
END_TYPE

// POUs/Controller/Lvl0/ECD (EtherCAT Diagnostic)/T_Ctrl_SIf_ECD_Cur
TYPE T_Ctrl_SIf_ECD_Cur :
STRUCT
	/// Shows the number of EtherCAT Slaves
	uinNumOfSlaves: UINT;
	/// Information of every slave
	stSlaveData: ARRAY[0..ECD_Const.cuinMaxSlaves] OF T_ECD_SlaveData;
	/// State Of Master
	worMasterState: WORD;
	/// All CRC Errors
	udiCRCSumm: UDINT;
	/// Counter of Slave Errors State
	uinNumOfSlaveErrors: UINT;
END_STRUCT
END_TYPE

// POUs/Controller/Lvl0/ECD (EtherCAT Diagnostic)/T_Ctrl_SIf_ECD_Par
TYPE T_Ctrl_SIf_ECD_Par :
STRUCT
	/// [ms] Timeout power on. Timeout for initialize all ADS connections.
	udiTOPowerOn_ms: UDINT;
	/// [ms] Timeout function over all slaves
	udiTOCheckAll_ms: UDINT;
	/// [ms] Timeout function for one slave
	udiTOCheckOne_ms: UDINT;
	/// [ms] Polling interval for States
	udiPollingInterval_ms: UDINT;
	/// Maximum CRC Value one slave 
	udiMaxCRC: UDINT;
END_STRUCT
END_TYPE

// POUs/Controller/Lvl0/ECD (EtherCAT Diagnostic)/T_ECD_SlaveData
TYPE T_ECD_SlaveData :
STRUCT
	/// Slave Configuration
	stConfigData: Tc2_EtherCAT.ST_EcSlaveConfigData;
	/// Address of the slave (as UINT, beacuase in stConfigData is only as WORD)
	uinAddress: UINT;
	/// State of the slave
	stState: Tc2_EtherCAT.ST_EcSlaveState;
	/// CRC Error totally
	stCRCError: Tc2_EtherCAT.ST_EcCrcErrorEx;
END_STRUCT
END_TYPE

// POUs/Controller/Lvl0/RFW (RFID Reader-Writer)/E_Typ_RFW
TYPE E_Typ_RFW :
(
	/// RF310
	RF310R := 0,
	/// RF382R
	RF382R := 1,
	Max_E_Typ_CYL
);
END_TYPE

// POUs/Controller/Lvl0/RFW (RFID Reader-Writer)/T_Ctrl_SIf_RFW
TYPE T_Ctrl_SIf_RFW :
STRUCT
	///configuration
	Cfg: T_Ctrl_SIf_RFW_Cfg;
	///parameter
	Par: T_Ctrl_SIf_RFW_Par;
	///current values
	Cur: T_Ctrl_SIf_RFW_Cur;
	///io input
	In: T_Ctrl_SIf_RFW_In;
	///io output
	Out: T_Ctrl_SIf_RFW_Out;
	///Data Channel from PLC to Line Controller
	DtChnToLine: T_Ctrl_SIf_RFW_DtChnToLine;	
	///alarm number used in this controller
	Alm: ARRAY[1..6] OF T_Ctrl_Alm;
END_STRUCT
END_TYPE

// POUs/Controller/Lvl0/RFW (RFID Reader-Writer)/T_Ctrl_SIf_RFW_Cfg
TYPE T_Ctrl_SIf_RFW_Cfg :
STRUCT
	eTyp: E_Typ_RFW;
	/// Get automatically the Tray ID too 
	bolGetTrayIDAuto: BOOL;
	/// Net ID oft EtherCat Master
	stNetId: TC2_SYSTEM.T_AmsNetID;
	/// Port Number of EtherCat Slave Comunication Module
	uinSlaveAddr: UINT;
	/// Send every New RFID to Line controller
	bolDtChToLine_send: BOOL;	
END_STRUCT
END_TYPE

// POUs/Controller/Lvl0/RFW (RFID Reader-Writer)/T_Ctrl_SIf_RFW_Cur
TYPE T_Ctrl_SIf_RFW_Cur :
STRUCT
	/// 1 = tag is present  
	bolPresent: BOOL;
	/// Data to read / write
	abytData: ARRAY[0..255] OF BYTE;
	/// Data in Structure
	stData: T_RFW;
	/// Job information, what data read or write
	dwoJob: DWORD;
END_STRUCT
END_TYPE

// POUs/Controller/Lvl0/RFW (RFID Reader-Writer)/T_Ctrl_SIf_RFW_DtChnToLine
TYPE T_Ctrl_SIf_RFW_DtChnToLine :
STRUCT
	stNewRfid: T_NewRFID_DtChn;
END_STRUCT
END_TYPE

// POUs/Controller/Lvl0/RFW (RFID Reader-Writer)/T_Ctrl_SIf_RFW_In
TYPE T_Ctrl_SIf_RFW_In :
STRUCT
END_STRUCT
END_TYPE

// POUs/Controller/Lvl0/RFW (RFID Reader-Writer)/T_Ctrl_SIf_RFW_Out
TYPE T_Ctrl_SIf_RFW_Out :
STRUCT
END_STRUCT
END_TYPE

// POUs/Controller/Lvl0/RFW (RFID Reader-Writer)/T_Ctrl_SIf_RFW_Par
TYPE T_Ctrl_SIf_RFW_Par :
STRUCT
	///[ms] until failure to long time for read
	udiReadTime_ms: UDINT;
	///[ms] until failure to long time for write
	udiWriteTime_ms: UDINT;
	///[ms] minimum wait time between two read command
	udiMinCmdTime: UDINT;
	///[ms] locktime prevents sending same ID's to LineControl multiple times
	udiLockTime: UDINT;
END_STRUCT
END_TYPE

// POUs/Controller/Lvl0/RFW (RFID Reader-Writer)/T_NewRFID_DtChn
TYPE T_NewRFID_DtChn :
STRUCT
	// new RF ID
	strID: STRING;			// configurable if Tag or Tray ID
	uliTagID: ULINT;
	strTimestamp: STRING(24);
	intDataState: INT;	
END_STRUCT
END_TYPE

// POUs/Controller/Lvl0/RFW (RFID Reader-Writer)/T_RFW
TYPE T_RFW :
STRUCT
	///	Repeteition ID			Identifies the try number in the sequence	
	usiRepetitionID: USINT;
	///	Workstation		2 workstations in the cell	1 BIT	0: Workstation1, 2: Workstation2
	bolWorkstation2: BOOL;
	///usiProductID : USINT;				// 	The product ID bits 1 to 5 are indeed not used. Mail T.Bosgiraud 11.6.2013 Product type	Max number of product types = 32	5 bits,	product ID (bits 1 to 5), 
	bolDeleteFileAfterPrint: BOOL;
	/// 	1 means that the image has been printed without problem.
	bolPrintOk: BOOL;
	///	0: Use the bottom of the tray as basis and add Offset
	bolHeightUseMeasure: BOOL;
	///	Email 1.06.2013 Berk “Use measured height=1”, the actual measurement of the  laser plus any offsets programmed into the tray are used to adjust the lifting height
	///	1: Use the printable product surface as basis and add Offset to the measured height
	usiHeightOffset: USINT;
	/// 	“Offset +/-” = 1 means that the printable surface OF the item will go further away FROM the print head.
	bolHeightOffsetSignMinus: BOOL;
	/// 	“Offset +/-” = 0 (default value) means that the printable surface of the item will come closer to the print head
	bolIonizer: BOOL;
	/// 	Pre-treatment	Plasma 0: Plasma off, 1: Level 1 ..3:Level3
	usiPlasmaLevel: USINT;
	/// 	Print numbers 1 means that the image needs to be printed twice on the products
	bolPrintPass: BOOL;
	/// 	1 means that the nozzle check pattern has to be printed onto the products.
	bolNozzleCheck: BOOL;
	///	1 means that the alignment check pattern has to be printed onto the products.
	bolAligneCheck: BOOL;
	///	UV-pinning intensity 0: Level1 ... 15: Level16
	usiUVPinningLevel: USINT;
	///	UV-lamp intensity 0: Level1 ... 15: Level16
	usiUVLampLevel: USINT;
	/// p.e.: 268205625-3.pdf -> The file name sent by VIPER to the printer and to the conveyor is made out of 64 bits
	strFileName: STRING;
	/// The RFID divides the rest of the name (268205625-3) as 8 successive bytes arranged as follows:
	///	-	Byte 7 (RFID byte 0Dhex) to byte 1 (RFID byte 07hex) express the number before the hyphen sign (in this case 268205625)
	///	-	Byte 0 (RFID byte 06hex) expresses the number after the hyphen sign (in this case 3).
	bolBrush: BOOL;
	///	1: use second brush means that the brush has TO be used FOR the considered tray
	bolBrushClean: BOOL;
	///	“Brush Fans”=1 means that the fans have to be used for the considered tray
	bolBrushFans: BOOL;
	///	“Gutter Clean”=1 means that the tray is running for gutter cleaning purposes.
	bolGutterClean: BOOL;
	/// 	This bit tells whether the tray is a regular production tray or a special tray (nozzle check, alignment...).
	bolSpecialTray: BOOL;
	/// 	Byte 0-13	->9999999999999	
	strTrayID: STRING;
	/// 	Byte 0-13	->9999999999999	
	strTagID: STRING;
	uliTagID: ULINT;
END_STRUCT
END_TYPE

// POUs/Controller/Lvl0/SGT (Signal Tower)/E_ALM_SGT
{attribute 'qualified_only' := ''}
TYPE E_ALM_SGT :
(
	Dummy := 1,
	MAX_E_ALM
) UINT;
END_TYPE

// POUs/Controller/Lvl0/SGT (Signal Tower)/T_Ctrl_SIf_SGT
TYPE T_Ctrl_SIf_SGT :
STRUCT
	/// configuration
	Cfg: T_Ctrl_SIf_SGT_Cfg;
	/// parameter
	Par: T_Ctrl_SIf_SGT_Par;
	/// io output
	Out: T_Ctrl_SIf_SGT_Out;
	/// alarm number used in this controller
	Alm: ARRAY[1..(E_ALM_SGT.MAX_E_ALM - 1)] OF T_Ctrl_Alm;
END_STRUCT
END_TYPE

// POUs/Controller/Lvl0/SGT (Signal Tower)/T_Ctrl_SIf_SGT_Cfg
TYPE T_Ctrl_SIf_SGT_Cfg :
STRUCT
	/// Enable lamp test in PONBusy state
	bolEnableLampTest: BOOL;
END_STRUCT
END_TYPE

// POUs/Controller/Lvl0/SGT (Signal Tower)/T_Ctrl_SIf_SGT_Out
TYPE T_Ctrl_SIf_SGT_Out :
STRUCT
	/// green lamp
	bolGreen: T_Ctrl_IoBool;
	/// yellow lamp
	bolYellow: T_Ctrl_IoBool;
	/// red lamp
	bolRed: T_Ctrl_IoBool;
	/// acoustic signal
	bolBeep: T_Ctrl_IoBool;
END_STRUCT
END_TYPE

// POUs/Controller/Lvl0/SGT (Signal Tower)/T_Ctrl_SIf_SGT_Par
TYPE T_Ctrl_SIf_SGT_Par :
STRUCT
	/// [ms] Blink interval time
	udiBlinkTime_ms: UDINT;
	/// [ms] Beep on time
	udiBeepOnTime_ms: UDINT;
	/// [ms] Beep off time
	udiBeepOffTime_ms: UDINT;
	/// [ms] Lamp test time, used in PONBusy
	udiLampTestTime_ms: UDINT;
END_STRUCT
END_TYPE

// POUs/Controller/Lvl0/UMC [Universal Motor Controller]/E_ALM_UMC
TYPE E_ALM_UMC :
(
	MotorOnTimeout 					:= 1,
	MotorError						:= 2,
	MotorWarning					:= 3,
	MotorOverCurrent				:= 4,
	MotorNotReady					:= 5,
	DirectionParameterOverflow		:= 6,
	SpeedOverLimit					:= 7,
	MAX_E_ALM_UMC
);
END_TYPE

// POUs/Controller/Lvl0/UMC [Universal Motor Controller]/E_CFG_UMC
TYPE E_CFG_UMC :
(
	Standard					:= 0,
	LenzeFC						:= 1,
	MAY_E_CFG_UMC
);
END_TYPE

// POUs/Controller/Lvl0/UMC [Universal Motor Controller]/E_TURN_DIRECTION
TYPE E_TURN_DIRECTION :
(
	AUTOMATIC		:= 0,
	LEFT			:= 1,
	RIGHT			:= 2,
	MAX_E_TURN_DIRECTION
);
END_TYPE

// POUs/Controller/Lvl0/UMC [Universal Motor Controller]/E_UMC_MOTOR_STATUS
TYPE E_UMC_MOTOR_STATUS :
(
	FirmwareUpdate 		:= 0,
	Init				:= 1,
	MotorIdent			:= 2,
	ReadyToSwitchON		:= 3,
	SwitchedON			:= 4,
	OperationEnabled	:= 5,
	Warning				:= 6,
	Trouble				:= 7,
	Fault				:= 8,
	TroubleQSP			:= 9,
	SafeTorqueOff		:= 10,
	SystemFail			:= 11,
	MAX_E_UMC_MOTOR_STATUS
);
END_TYPE

// POUs/Controller/Lvl0/UMC [Universal Motor Controller]/T_Ctrl_SIf_UMC
TYPE T_Ctrl_SIf_UMC :
STRUCT
	///configuration
	Cfg: T_Ctrl_SIf_UMC_Cfg;
	///parameter
	Par: T_Ctrl_SIf_UMC_Par;
	///current values
	Cur: T_Ctrl_SIf_UMC_Cur;
	///io input
	In: T_Ctrl_SIf_UMC_In;
	///io output
	Out: T_Ctrl_SIf_UMC_Out;
	///alarm number used in this controller
	Alm: ARRAY[1..MAX_E_ALM_UMC] OF T_Ctrl_Alm;
	///interlock of output/movements
	Ilk: T_Ctrl_SIf_UMC_Ilk;
END_STRUCT
END_TYPE

// POUs/Controller/Lvl0/UMC [Universal Motor Controller]/T_Ctrl_SIf_UMC_Cfg
TYPE T_Ctrl_SIf_UMC_Cfg :
STRUCT
	/// Motor Type
	MotorType							: E_CFG_UMC;			
	/// [RPM] L0011 Setting of the Lenze motor. This value is 100% of the output control setting.
	uinLC11								: UINT;
	/// Value that is equal to 100% of LC11
	uinLC11_100							: UINT;
	/// Maximum allowed speed in [%] of LC11
	uinMaxSpeed							: UINT;
END_STRUCT
END_TYPE

// POUs/Controller/Lvl0/UMC [Universal Motor Controller]/T_Ctrl_SIf_UMC_Cur
TYPE T_Ctrl_SIf_UMC_Cur :
STRUCT	
	/// Actual Turning Direction
	eDirection								: E_TURN_DIRECTION;
	/// Actual speed as output 16384 = 100% of L-C11 (1500RPM)
	uinSpeedOuput							: UINT;
	/// Actual speed as output in [rpm]
	uinSpeed_rpm							: UINT;
	/// Motor Limit as Output value
	uinSpeedLimit							: UINT;
	/// Motor reset retries
	uinMotorResetCnt					: UINT;
END_STRUCT
END_TYPE

// POUs/Controller/Lvl0/UMC [Universal Motor Controller]/T_Ctrl_SIf_UMC_Ilk
TYPE T_Ctrl_SIf_UMC_Ilk :
STRUCT
END_STRUCT
END_TYPE

// POUs/Controller/Lvl0/UMC [Universal Motor Controller]/T_Ctrl_SIf_UMC_In
TYPE T_Ctrl_SIf_UMC_In :
STRUCT
	/// Status Word of Lenze
	uinStatus				: Base_PLC.T_Ctrl_IoUint;
	/// Motor actual speed
	intMotorActualSpeed		: Base_PLC.T_Ctrl_IoInt;
	/// Motor actual speed setpoint 
	uinMotorSetSpeed		: Base_PLC.T_Ctrl_IoUint;
	/// Is the EMO Ok...
	bolEmoOk				: Base_PLC.T_Ctrl_IoBool;
END_STRUCT
END_TYPE

// POUs/Controller/Lvl0/UMC [Universal Motor Controller]/T_Ctrl_SIf_UMC_Out
TYPE T_Ctrl_SIf_UMC_Out :
STRUCT
	/// Control word for Lenze FU
	uinControl			: BASE_PLC.T_Ctrl_IoUint;
	/// Speed Setpoint; 16384 (214) ≡ 100% (bez. auf L-C11)
	uinSpeedSetpoint	: BASE_PLC.T_Ctrl_IoUint;
END_STRUCT
END_TYPE

// POUs/Controller/Lvl0/UMC [Universal Motor Controller]/T_Ctrl_SIf_UMC_Par
TYPE T_Ctrl_SIf_UMC_Par :
STRUCT
	/// Rotation direction E_CFG_UMC
	eRotationDirection					: E_TURN_DIRECTION;
	/// [ms] time to initialize and reset the errors on the motor
	udiStartupOnTime_ms					: UDINT;
	/// [ms] time the motor has time to go from OFF to ON
	udiMotorOnTime_ms					: UDINT;
	/// [rpm] Speed control selection
	uinSpeed_rpm						: UINT;
	/// [ms] time to wait until the motor reaches the set speed.
	udiSimMotorOnTime_ms				: UDINT;
	/// [ms] Delay until the drive startsup
	udiMoveStartLatency					: UDINT;
	/// [ms] Delay until the drive stops 
	udiMoveStopLatency					: UDINT;
	/// Motor reset retries
	uinMotorResetCnt					: UINT;
	// [ms] Motor Reset Pulse Time		
	uinMotorResetPulseTime_ms			: UINT;
END_STRUCT
END_TYPE

// POUs/Controller/Lvl0/UMC [Universal Motor Controller]/T_UMC_Lenze_Control
TYPE T_UMC_Lenze_Control :
STRUCT
	SwitchOn		: BIT;
	DisableVoltage	: BIT;
	SetQuickStop	: BIT;
	EnableOperation	: BIT;
	ModeSpecific_1  : BIT;
	ModeSpecific_2  : BIT;
	ModeSpecific_3  : BIT;
	ResetFault		: BIT;
	SetHalt			: BIT;
	Reserved_1 		: BIT;
	Reserved_2		: BIT;
	SetDCBreak		: BIT;
	JogSpeed1		: BIT;
	JogSpeed2		: BIT;
	SetFail			: BIT;
	SetSpeedCcw		: BIT;
END_STRUCT
END_TYPE

// POUs/Controller/Lvl0/UMC [Universal Motor Controller]/T_UMC_Lenze_Status
TYPE T_UMC_Lenze_Status :
STRUCT
	FreeStatusBit0			: BIT;
	PowerDisabled_IMP		: BIT;
	ImaxActive				: BIT;
	SpeedSetReached			: BIT;
	SpeedActEqualSet		: BIT;
	NActualCompare			: BIT;
	ActSpeedIsZero			: BIT;
	ControllerInhibit		: BIT;
	Status_1				: BIT;
	Status_2				: BIT;
	Status_3				: BIT;
	Status_4				: BIT;
	Warning					: BIT;
	Trouble					: BIT;
	SpeedCcw				: BIT;
	DriveReady				: BIT;
END_STRUCT
END_TYPE

// POUs/Controller/Lvl0/UMC [Universal Motor Controller]/U_UMC_Lenze_Control
TYPE U_UMC_Lenze_Control :
UNION
	Output		: UINT;
	Data		: T_UMC_Lenze_Control;
END_UNION
END_TYPE

// POUs/Controller/Lvl0/UMC [Universal Motor Controller]/U_UMC_Lenze_Status
TYPE U_UMC_Lenze_Status :
UNION
	Input		: UINT;	
	Data		: T_UMC_Lenze_Status;
END_UNION
END_TYPE

// POUs/Controller/Lvl0/VLV (Valve controller)/E_ALM_VLV
{attribute 'qualified_only' := ''}
TYPE E_ALM_VLV :
(
	SensorOpenAlwaysOn := 1,
	SensorCloseNotReached := 2,
	SensorCloseAlwaysOn := 3,
	SensorOpenNotReached := 4,
	InterlockOpen := 5,
	InterlockClose := 6,
	MAX_E_ALM
) UINT;
END_TYPE

// POUs/Controller/Lvl0/VLV (Valve controller)/E_Typ_VLV
TYPE E_Typ_VLV :
(
	///bistabile and two feedback sensors
	Valve2_Sensor2 := 0,
	///bistabile and open feedback sensor	
	Valve2_SensorOpened,
	///bistabile and close feedback sensor
	Valve2_SensorClosed,
	///bistabile and no feedback sensors
	Valve2_Sensor0,
	///monostabile and 2 feedback sensors	
	Valve1_Sensor2,
	///monostabile and open feedback sensor	
	Valve1_SensorOpened,
	///monostabile and close feedback sensor
	Valve1_SensorClosed,
	///monostabile and no feedback sensors
	Valve1_Sensor0,
	Max_E_Typ_VLV
);
END_TYPE

// POUs/Controller/Lvl0/VLV (Valve controller)/T_Ctrl_SIf_VLV
TYPE T_Ctrl_SIf_VLV :
STRUCT
	///configuration
	Cfg: T_Ctrl_SIf_VLV_Cfg;
	///parameter
	Par: T_Ctrl_SIf_VLV_Par;
	///current values
	Cur: T_Ctrl_SIf_VLV_Cur;
	///io input
	In: T_Ctrl_SIf_VLV_In;
	///io output
	Out: T_Ctrl_SIf_VLV_Out;
	///alarm number used in this controller
	Alm: ARRAY[1..(E_ALM_VLV.MAX_E_ALM - 1)] OF T_Ctrl_Alm;
	///interlock of output/movements
	Ilk: T_Ctrl_SIf_VLV_Ilk;
END_STRUCT
END_TYPE

// POUs/Controller/Lvl0/VLV (Valve controller)/T_Ctrl_SIf_VLV_Cfg
TYPE T_Ctrl_SIf_VLV_Cfg :
STRUCT
	eTyp: E_Typ_VLV;
END_STRUCT
END_TYPE

// POUs/Controller/Lvl0/VLV (Valve controller)/T_Ctrl_SIf_VLV_Cur
TYPE T_Ctrl_SIf_VLV_Cur :
STRUCT
	///[ms] time last movement to open	
	udiMoveTimeOpen: UDINT;
	///[ms] time last movement to close
	udiMoveTimeClose: UDINT;
END_STRUCT
END_TYPE

// POUs/Controller/Lvl0/VLV (Valve controller)/T_Ctrl_SIf_VLV_Ilk
TYPE T_Ctrl_SIf_VLV_Ilk :
STRUCT
	///interlock open valve
	bolOpen: BOOL;
	///interlock close valve
	bolClose: BOOL;
END_STRUCT
END_TYPE

// POUs/Controller/Lvl0/VLV (Valve controller)/T_Ctrl_SIf_VLV_In
TYPE T_Ctrl_SIf_VLV_In :
STRUCT
	///sensor feedback position open reached
	bolOpen: T_Ctrl_IoBool;
	///sensor feedback position close reached
	bolClose: T_Ctrl_IoBool;
END_STRUCT
END_TYPE

// POUs/Controller/Lvl0/VLV (Valve controller)/T_Ctrl_SIf_VLV_Out
TYPE T_Ctrl_SIf_VLV_Out :
STRUCT
	///switch valve open
	bolOpen: T_Ctrl_IoBool;
	///switch valve close
	bolClose: T_Ctrl_IoBool;
END_STRUCT
END_TYPE

// POUs/Controller/Lvl0/VLV (Valve controller)/T_Ctrl_SIf_VLV_Par
TYPE T_Ctrl_SIf_VLV_Par :
STRUCT
	///[ms] until failure to long time for open	
	udiOpenTime_ms: UDINT;
	///[ms] until failure to long time for close	
	udiCloseTime_ms: UDINT;
	///[ms] simulation time for open or /2 of timeout time?
	udiSimOpenTime_ms: UDINT;
	///[ms] simulation time for close or /2 of timeout time?
	udiSimCloseTime_ms: UDINT;
END_STRUCT
END_TYPE

// POUs/Controller/Lvl0/VPC [Vacuum Pump Controller]/E_ALM_VPC
TYPE E_ALM_VPC :
(
	VacuumPumpOnTimeout 	:= 1,
	VacuumPumpOffTimeout	:= 2,
	VacuumFailure			:= 3,
	MAX_E_ALM_VPC
);
END_TYPE

// POUs/Controller/Lvl0/VPC [Vacuum Pump Controller]/E_CFG_VPC
TYPE E_CFG_VPC :
(
	/// Only Vacuum Motor with no feedback
	Standard					:= 0,
	VaccumSensor				:= 1,
	MotorFeedback				:= 2,
	MAY_E_CFG_CYL
);
END_TYPE

// POUs/Controller/Lvl0/VPC [Vacuum Pump Controller]/T_Ctrl_SIf_VPC
TYPE T_Ctrl_SIf_VPC :
STRUCT
	///configuration
	Cfg: T_Ctrl_SIf_VPC_Cfg;
	///parameter
	Par: T_Ctrl_SIf_VPC_Par;
	///current values
	Cur: T_Ctrl_SIf_VPC_Cur;
	///io input
	In: T_Ctrl_SIf_VPC_In;
	///io output
	Out: T_Ctrl_SIf_VPC_Out;
	///alarm number used in this controller
	Alm: ARRAY[1..E_ALM_VPC.MAX_E_ALM_VPC] OF T_Ctrl_Alm;
	///interlock of output/movements
	Ilk: T_Ctrl_SIf_VPC_Ilk;
END_STRUCT
END_TYPE

// POUs/Controller/Lvl0/VPC [Vacuum Pump Controller]/T_Ctrl_SIf_VPC_Cfg
TYPE T_Ctrl_SIf_VPC_Cfg :
STRUCT
	VacuumPumpFeedback			: BOOL;				// VacuumPump has a feedback
	VacuumSensorAvailable		: BOOL;				// Vacuum Sensor available
END_STRUCT
END_TYPE

// POUs/Controller/Lvl0/VPC [Vacuum Pump Controller]/T_Ctrl_SIf_VPC_Cur
TYPE T_Ctrl_SIf_VPC_Cur :
STRUCT	
END_STRUCT
END_TYPE

// POUs/Controller/Lvl0/VPC [Vacuum Pump Controller]/T_Ctrl_SIf_VPC_Ilk
TYPE T_Ctrl_SIf_VPC_Ilk :
STRUCT
END_STRUCT
END_TYPE

// POUs/Controller/Lvl0/VPC [Vacuum Pump Controller]/T_Ctrl_SIf_VPC_In
TYPE T_Ctrl_SIf_VPC_In :
STRUCT
	/// 0 = Vacuum is NOK; 1 = Vacuum is Ok --> Vacuum Pump is probably running
	bolVacuumOk				: BASE_PLC.T_Ctrl_IoBool;
	/// Pump has a feedback
	bolPumpOn				: BASE_PLC.T_Ctrl_IoBool;
END_STRUCT
END_TYPE

// POUs/Controller/Lvl0/VPC [Vacuum Pump Controller]/T_Ctrl_SIf_VPC_Out
TYPE T_Ctrl_SIf_VPC_Out :
STRUCT
	/// 0 = Vacuum Pump Off; 1 = Vacuum Pump On
	bolVacuumPumpOn			: BASE_PLC.T_Ctrl_IoBool;
END_STRUCT
END_TYPE

// POUs/Controller/Lvl0/VPC [Vacuum Pump Controller]/T_Ctrl_SIf_VPC_Par
TYPE T_Ctrl_SIf_VPC_Par :
STRUCT
	/// [ms] time the pump has time to go from OFF to ON
	udiVacuumPumpTime_ms				: UDINT;
	/// [ms] vacuum stabilization time if no vacuum sensor is available
	udiVacuumStabilizationTime_ms		: UDINT;
	/// [ms] time to wait until the vacuum sensor off is acknowledged as off.
	udiVacuumSensorDebounceTime_ms		: UDINT;
	/// [ms] simulation time for Vacuum Pump ON
	udiSimVacuumPumpOnTime_ms			: UDINT;
END_STRUCT
END_TYPE

// POUs/Controller/Lvl3/BaseCtrlModule/T_Ctrl_SIf_MOD
TYPE T_Ctrl_SIf_MOD :
STRUCT
	/// configuration
	Cfg: POINTER TO T_Ctrl_SIf_MOD_Cfg;
	/// parameter
	Par: POINTER TO T_Ctrl_SIf_MOD_Par;
	/// current values
	Cur: POINTER TO T_Ctrl_SIf_MOD_Cur;
	/// io input
	In: POINTER TO T_Ctrl_SIf_MOD_In;
	/// alarm number used in this controller
	Alm: ARRAY[1..6] OF T_Ctrl_Alm;
END_STRUCT
END_TYPE

// POUs/Controller/Lvl3/BaseCtrlModule/T_Ctrl_SIf_MOD_Cfg
TYPE T_Ctrl_SIf_MOD_Cfg :
STRUCT
	/// Enable communication to line control
	bolComToLineControlEnabled: BOOL;
END_STRUCT
END_TYPE

// POUs/Controller/Lvl3/BaseCtrlModule/T_Ctrl_SIf_MOD_Cur
TYPE T_Ctrl_SIf_MOD_Cur :
STRUCT
	/// Max module capacity calculated from all childs which implement interface IBuffer
	dinMaxCapacity: DINT;
	/// Actual number of hangers calculated from all childs which implement interface IBuffer
	dinNumOfHangers: DINT;
	/// Togglebit to Line Control
	bolKeepAliveHost: BOOL;
	bolKeepAlivePlc: BOOL;
	/// LineControl-Signal: Input Buffer is Full
	a_bBufferIsFull: ARRAY[0..10] OF BOOL;
	/// LineControl-Signal: If true Module is not allowed to release hangers (but can be still in RUN state). 
	bolStopReleaseHangers: BOOL;
END_STRUCT
END_TYPE

// POUs/Controller/Lvl3/BaseCtrlModule/T_Ctrl_SIf_MOD_In
TYPE T_Ctrl_SIf_MOD_In :
STRUCT
	/// Inputs from global module for general supervision 
	/// Emergency circuit ok
	bolEmergencyOffOk: T_Ctrl_IoBool;
	/// No general error active, will be set to FALSE if there is an global error like e.g. over temperature in cabinet. 
	bolNoGeneralError: T_Ctrl_IoBool;
END_STRUCT
END_TYPE

// POUs/Controller/Lvl3/BaseCtrlModule/T_Ctrl_SIf_MOD_Par
TYPE T_Ctrl_SIf_MOD_Par :
STRUCT
	/// [ms] Communication timeout to line control
	udiComTimeOutLineCtrl_ms: UDINT;
	/// [ms] Array with wait time for run groups
	aListOfRunGrpWaitTime_ms: ARRAY[0..Base_Const.cMaxNrOfChilds] OF UDINT;
	/// [ms] Array with wait time for stop groups
	aListOfStopGrpWaitTime_ms: ARRAY[0..Base_Const.cMaxNrOfChilds] OF UDINT;
	/// [ms] timeout for stopping (0= disable timeout monitoring)
	udiTimeoutStopping_ms: UDINT;
	/// [ms] timeout for starting (0= disable timeout monitoring)
	udiTimeoutStarting_ms: UDINT;
END_STRUCT
END_TYPE

// POUs/Controller/Lvl3/BaseCtrlModule/T_Sequence
TYPE T_Sequence :
STRUCT
	pChild: POINTER TO fb_CtrlBase;
	/// Access to CIF of child
	pCIF: POINTER TO T_Ctrl_CIf;
	/// Associated run sequence group
	uinGroupRun: UINT;
	/// Associated stop sequence group
	uinGroupStop: UINT;
	/// Command to be executed for run sequence
	intCmdSeqRun: INT;
	/// Expected status for run sequence
	intStatusSeqRun: INT;
	/// Alternativ status for run sequence
	intStatusSeqRun2: INT;
	/// Command to be executed for run sequence
	intCmdSeqStop: INT;
	/// Expected status for run sequence
	intStatusSeqStop: INT;
	/// Used internal for run and stop sequence to detect if the sequence has been processed
	bolChecked: BOOL;
END_STRUCT
END_TYPE

// POUs/Utility/Data Channel/IdBase/T_IdBaseRecvData
TYPE T_IdBaseRecvData :
STRUCT
	fbDataChannel						: FB_IdBaseRecvDch;
	rDataChannelItem					: T_IdBase_DCH;
	fbFifo								: FB_DataChannelRecvFifo;
	rFifoItem							: T_IdBase_DCH;
	aFifoBuffer							: ARRAY [0..cRECVDATACHANNELBUFFER-1] OF T_IdBase_DCH;
END_STRUCT
END_TYPE

// POUs/Utility/Data Channel/IdBase/T_IdBaseSendData
TYPE T_IdBaseSendData :
STRUCT
	fbDataChannel						: FB_IdBaseSendDch;
	rDataChannelItem					: T_IdBase_DCH;
	fbFifo								: FB_DataChannelSenderFifo;
END_STRUCT
END_TYPE

// POUs/Utility/DCH [Data Channel Base]/E_DCH_Error
TYPE E_DCH_Error :
(
	None,
	Unknown,
	MAX_E_DCH_Error
);
END_TYPE

// POUs/Utility/DCH [Data Channel Base]/E_PlcSaberDHCState
TYPE E_PlcSaberDHCState :
(
	Init,						// 0
	WaitForJob,					// 1
	SendData,					// 2
	Acknowledge,				// 3
	Retry,						// 4
	Error,						// 5
	WaitChannelInit,			// 6
	MAX_E_PlcSaberDHCStat
);
END_TYPE

// POUs/Utility/DCH [Data Channel Base]/E_SaberPlcDHCState
TYPE E_SaberPlcDHCState :
(
	Init,						// 0
	WaitForData,				// 1
	RecvData,					// 2
	DataReady,					// 3
	Acknowledge,				// 4
	Retry,						// 5
	Error,						// 6
	WaitChannelInit,			// 7
	MAX_E_PlcSaberDHCStat
);
END_TYPE

// POUs/Utility/GHT [Generic Hash Table]/T_GHTHashTableBuffer
TYPE T_GHTHashTableBuffer :
STRUCT
	aBuffer		: ARRAY[0..50-1] OF POINTER TO T_HashTableEntry;	
END_STRUCT
END_TYPE

// POUs/Utility/ItemBase/E_Destination
TYPE E_Destination :
(
	StackerA,
	StackerB,
	StackerC,
	Garbage,
	MAX_E_Destination
);
END_TYPE

// POUs/Utility/ItemBase/E_ItemHealth
TYPE E_ItemHealth :
(
	Healthy,							// 0
	Ovn_Temperature,					// 1
	Ovn_Time,							// 2
	Ovn_Lost,							// 3
	Hpm_Time,							// 4
	Hpm_Pressure,						// 5
	Hpm_Temperature,					// 6
	Hpm_Lost,							// 7
	Hpm_Unknown,						// 8
	Failed,								// 9
	Lost,								// 10	- Item is lost somewhere	
	MAX_E_ItemHealth
);
END_TYPE

// POUs/Utility/ItemBase/E_PrintSelection
TYPE E_PrintSelection :
(
	// Binary Enum. Print A&B = PrintHeadA | PrintHeadB = 0x03
	None		 	:= 16#00,
	PrintHeadA		:= 16#01,
	PrintHeadB		:= 16#02,
	MAX_E_PrintSelection
);
END_TYPE

// POUs/Utility/ItemBase/T_IdBase_DCH
{attribute 'enable_dynamic_creation'}
//{attribute 'pack_mode' := '1'}
TYPE T_IdBase_DCH:
STRUCT
	rBaseInfo					: T_ItemBase;
	// Real read process ID values
	udiIdentification			: ULINT;	
END_STRUCT
END_TYPE

// POUs/Utility/ItemBase/T_ItemBase
{attribute 'enable_dynamic_creation'}
//{attribute 'pack_mode' := '1'}
TYPE T_ItemBase :
STRUCT
	// Item Empty
	bolItemAvailable			: BOOL;
	
	// Actual Status of the item.
	eHealth						: E_ItemHealth 		:= E_ItemHealth.Healthy;
	
	// Actual Position
	uinModuleId					: UINT;
	uinActualPosition			: UINT;
	
	dtStartTimeStamp			: TC2_UTILITIES.TIMESTRUCT;
END_STRUCT
END_TYPE

// POUs/Utility/ItemBase/T_ItemPaperBase
{attribute 'enable_dynamic_creation'}
//{attribute 'pack_mode' := '1'}
TYPE T_ItemPaperBase EXTENDS T_ItemBase :
STRUCT
	// Real read process ID values
	udiPaperIdProcess			: UDINT;		// Paper ID
	// Set Value of the ID
	udiPaperIdSet				: UDINT;		// Paper ID
	// true if this is the paper is the last of a stack. After this paper is placed the stack is ejected.
	bolLastPaperOfStackBatch	: UINT;			
	// [ms] Time difference to the previous Paper
	udiDifferenceToPrevious_ms	: UDINT;
	// [ms] Time difference to the next paper
	udiDifferenceToNext_ms		: UDINT;
	// Paper Stream Destination
	eDestination				: E_Destination;
END_STRUCT
END_TYPE

// POUs/Utility/ItemBase/T_QueueBase
{attribute 'enable_dynamic_creation'}
//{attribute 'pack_mode' := '1'}
TYPE T_QueueBase :
STRUCT
	pData			: POINTER TO BYTE;	
	pNext			: POINTER TO T_QueueBase;
	pPrevious		: POINTER TO T_QueueBase;
END_STRUCT
END_TYPE

// POUs/Controller/Driver/ACL (ADS client for data exchange)/ACL_Const
VAR_GLOBAL CONSTANT
	cuinMaxConnections: UINT := 50;
END_VAR

// POUs/Controller/Driver/ACL (ADS client for data exchange)/ADS_IndexGroup
VAR_GLOBAL CONSTANT
	/// "Index-Group/Offset", GET_SYMHANDLE_BYNAME
	cGET_SYMHANDLE_BYNAME: UDINT := 16#F003;
	/// "Index-Group/Offset", READ_WRITE_SYMVAL_BYHANDLE
	cREAD_WRITE_SYMVAL_BYHANDLE: UDINT := 16#F005;
END_VAR

// POUs/Controller/Driver/BCD (Bar code driver)/BCD_CmdState
VAR_GLOBAL CONSTANT
	/// ctrl commands definitions
	cBCD_CMD_DONE: INT := -1;
	/// Connect TCP socket
	cBCD_CMD_CONNECT_SOCKET: INT := 1002;
	/// Close TCP socket
	cBCD_CMD_CLOSE_SOCKET: INT := 1004;
	/// Communication test 
	cBCD_CMD_COM_TEST: INT := 1006;
	/// Readout device information
	cBCD_CMD_READ_DEV_INFO: INT := 1008;
	/// Readout operating data
	cBCD_CMD_READ_OP_DATA: INT := 1010;
	/// Readout service information	
	cBCD_CMD_READ_SERVICE_INFO: INT := 1012;
	/// Command enable the sensor gate for X-TIME ("duration" setting of sensor object trigger)
	cBCD_CMD_READ_BARCODE: INT := 1014;
	/// Sensor try to detect a barcode.
	/// ctrl state definitions
	cBCD_STA_WaitForJob: INT := 1000;
	/// Open TCP socket busy
	cBCD_STA_ConnectSocketBusy: INT := 1002;
	/// Close TCP socket busy
	cBCD_STA_CloseSocketBusy: INT := 1004;
	/// TCP socket closed
	cBCD_STA_SocketClosed: INT := 1006;
	/// Communication test busy
	cBCD_STA_ComTestBusy: INT := 1008;
	/// Read bar code busy
	cBCD_STA_ReadCodeBusy: INT := 1010;
	/// Error
	cBCD_STA_Error: INT := 256;
END_VAR

// POUs/Controller/Driver/PRS [Present Sensor]/PRS_CmdState
VAR_GLOBAL CONSTANT
	///ctrl commands definitions
	///specific commands >200 - every command has to be a even number
;
	///ctrl specific states definitions
	cSTA_PRESENTBusy  			: INT := 201;
	cSTA_PRESENT      			: INT := 202;
	cSTA_ABSENTBusy 			: INT := 203;
	cSTA_ABSENT			     	: INT := 204;
END_VAR

// POUs/Controller/Driver/RFD (RFID Driver)/RFD_Cmd
VAR_GLOBAL CONSTANT
	/// ctrl state definitions
	/// Error
	cRFD_STA_Error: INT := 256;
	/// Power On
	cRFD_STA_PowerOnBusy: INT := 999;
	cRFD_STA_WaitForJob: INT := 1002;
	/// RESET Reader 
	cRFD_STA_ResetBusy: INT := 1003;
	/// Turn Off antenna 
	cRFD_STA_OffBusy: INT := 1007;
	cRFD_STA_Off: INT := 1008;
	/// Write Data to Tag 
	cRFD_STA_WriteBusy: INT := 1009;
	/// Read Data from Tag 
	cRFD_STA_ReadBusy: INT := 1011;
	/// Tag initialisation 
	cRFD_STA_TagInitBusy: INT := 1013;
	/// Check connection to antenna
	cRFD_STA_CheckBusy: INT := 1017;
	/// Service function read MDS-State (State of the near Tag)
	cRFD_STA_MDSBusy: INT := 1019;
	/// Service function read SLG State (State of the antenna)
	cRFD_STA_SLGBusy: INT := 1021;
	/// ctrl commands definitions
	/// specific commands >200 - every command has to be a even number
	cRFD_CMD_DONE: INT := -1;
	/// Switch controller on 
	cRFD_CMD_CTRL_ON: INT := 1000;
	/// Switch controller off 
	cRFD_CMD_CTRL_OFF: INT := 1006;
	/// Write Data to Tag 
	cRFD_CMD_Write: INT := 1010;
	/// Read Data from Tag 
	cRFD_CMD_Read: INT := 1012;
	/// Check connection to antenna 
	cRFD_CMD_Check: INT := 1018;
	/// Service function read MDS-State (State of the near Tag)
	cRFD_CMD_MDS: INT := 1020;
	/// Service function read SLG State (State of the antenna)
	cRFD_CMD_SLG: INT := 1022;
	/// Sub States
	/// Power On Busy
	cRFD_SUB_SetBaudrate: INT := 2001;
	/// Set Communication Settings
	cRFD_SUB_SetComSettings: INT := 2002;
	///  Clear Buffer
	cRFD_SUB_ClearBuffer: INT := 2003;
	/// Initialisation String sending
	cRFD_SUB_InitString: INT := 2004;
	///  Check Power On State
	cRFD_SUB_CheckPon: INT := 2005;
	/// OFF Busy
	cRFD_SUB_Prepare: INT := 2010;
	/// Data send
	cRFD_SUB_SendBusy: INT := 2011;
	/// Wait Answer
	cRFD_SUB_WaitAnswer: INT := 2012;
	/// SLG Write Mode 1
	cRFD_SUB_Write1: INT := 2020;
	/// SLG Wait Mode 1
	cRFD_SUB_Wait1: INT := 2021;
	/// SLG Write Mode 6
	cRFD_SUB_Write6: INT := 2022;
	/// SLG Wait Mode 6
	cRFD_SUB_Wait6: INT := 2023;
	///  Substates finished
	cRFD_SUB_SubStatesEnd: INT := 2100;
END_VAR

// POUs/Controller/Driver/RFD (RFID Driver)/RFD_Constants
VAR_GLOBAL
END_VAR

// POUs/Controller/Lvl0/BCC (Barcode controller)/BCC_CmdState
VAR_GLOBAL CONSTANT
	/// ctrl commands definitions
	/// specific commands >200 - every command has to be a even number
	cBCC_CMD_READ: INT := 202;
	/// ctrl specific states definitions
	cBCC_STA_READBusy: INT := 201;
	cBCC_STA_READ: INT := cBCC_CMD_READ;
END_VAR

// POUs/Controller/Lvl0/CYL (Cylinder)/CYL_CmdState
VAR_GLOBAL CONSTANT
	///ctrl commands definitions
	///specific commands >200 - every command has to be a even number
	cCMD_RETRACT: INT := 202;
	cCMD_EXTEND: INT := 204;
	///ctrl specific states definitions
	cSTA_RETRACTBusy: INT := 201;
	cSTA_RETRACT: INT := CYL_CmdState.cCMD_RETRACT;
	cSTA_EXTENDBusy: INT := 203;
	cSTA_EXTEND: INT := CYL_CmdState.cCMD_EXTEND;
END_VAR

// POUs/Controller/Lvl0/DRV (Drive)/Const_DRV
VAR_GLOBAL CONSTANT
	cMAX_BLOCKED_SUP: INT := 3;
END_VAR

// POUs/Controller/Lvl0/ECD (EtherCAT Diagnostic)/ECD_Const
VAR_GLOBAL CONSTANT
	cuinMaxSlaves: UINT := 256;
END_VAR

// POUs/Controller/Lvl0/RFW (RFID Reader-Writer)/RFID_Data
VAR_GLOBAL CONSTANT
	/// RFID Data connection
	/// See RFID Specification
	/// Defines the Start Adress and the lengh of the Data in the RF ID Tag
	/// Every DoubleWord has to Words, Higher is lengh, lower word is Startadress
	/// Example	
	/// 16#010005 => Startadress 5 Byte 1 => UV Settings
	cRFID_RepetionID: DWORD := 16#10100;
	cRFID_TrayInfo: DWORD := 16#10101;
	cRFID_HeighOfTray: DWORD := 16#10102;
	cRFID_Pretreatment: DWORD := 16#10103;
	cRFID_UVcuring: DWORD := 16#10104;
	cRFID_Filename: DWORD := 16#80105;
	cRFID_Brush: DWORD := 16#1010D;
	cRFID_TrayID: DWORD := 16#E0000;
	cRFID_TagID: DWORD := 16#8FFF0;
	cRFID_AllData: DWORD := 16#F0100;
END_VAR

// POUs/Controller/Lvl0/RFW (RFID Reader-Writer)/RFW_CmdState
VAR_GLOBAL CONSTANT
	///ctrl commands definitions
	///specific commands >200 - every command has to be a even number
	cCMD_ON: INT := 202;
	cCMD_READ: INT := 204;
	cCMD_WRITE: INT := 206;
	///ctrl specific states definitions
	cSTA_ONBusy: INT := 201;
	cSTA_ON: INT := cCMD_ON;
	cSTA_READBusy: INT := 203;
	cSTA_READ: INT := cCMD_READ;
	cSTA_WRITEBusy: INT := 205;
	cSTA_WRITE: INT := cCMD_WRITE;
END_VAR

// POUs/Controller/Lvl0/UMC [Universal Motor Controller]/UMC_CmdState
VAR_GLOBAL CONSTANT
	///ctrl commands definitions
	///specific commands >200 - every command has to be a even number
	cCMD_RIGHT				: INT := 202;
	cCMD_LEFT				: INT := 204;
	
	///ctrl specific states definitions
	cSTA_SETOPERATIONMODE	: INT := 201;
	cSTA_RESETMOTORERROR	: INT := 203;
END_VAR

// POUs/Controller/Lvl0/VLV (Valve controller)/VLV_CmdState
VAR_GLOBAL CONSTANT
	///ctrl commands definitions
	///specific commands >200 - every command has to be a even number
	cCMD_OPEN: INT := 202;
	cCMD_CLOSE: INT := 204;
	///ctrl specific states definitions
	cSTA_OPENBusy: INT := 201;
	cSTA_OPEN: INT := VLV_CmdState.cCMD_OPEN;
	cSTA_CLOSEBusy: INT := 203;
	cSTA_CLOSE: INT := VLV_CmdState.cCMD_CLOSE;
END_VAR

// POUs/Controller/Lvl0/VPC [Vacuum Pump Controller]/VPC_CmdState
VAR_GLOBAL CONSTANT
	///ctrl specific states definitions
	cSTA_VPC_StabilizeBusy: INT := 201;
END_VAR

// POUs/Utility/Data Channel/IdBase/IdBaseConst
VAR_GLOBAL CONSTANT
	cRECVDATACHANNELBUFFER 		:INT := 20;
END_VAR

// POUs/Utility/ItemBase/ItemConst
VAR_GLOBAL CONSTANT
	MAX_OVEN_SEGMENTS 				: UINT := 7;
	MAX_PRINT_HEAD_COUNT			: UINT := 5;
	MAX_PRINT_MODULE_COUNT			: UINT := 2;
END_VAR

// Version/Global_Version
// This function has been automatically generated from the project information.
VAR_GLOBAL CONSTANT
	{attribute 'const_non_replaced'}
	stLibVersion_Base_Elements : ST_LibVersion := (iMajor := 0, iMinor := 0, iBuild := 1, iRevision := 22, sVersion := '0.0.1.22');
END_VAR

// POUs/Controller/Driver/ACL (ADS client for data exchange)/FB_ACL
FUNCTION_BLOCK FB_ACL EXTENDS FB_CtrlBase
VAR
	// Specific interface struct for public access
	SIf: T_Ctrl_SIf_ACL;
	
	// Used blocks from lib. "utilities" for AMS route handling
	fbAddRoute:	FB_AddRouteEntry;
	
	// Used ADS blocks for communication
	fbWrite: ADSWRITE;
	fbRead: ADSREAD;
	fbReadWrite: ADSRDWRT;
		
	// List of all ADS connections handled by this block
	aListOfConnections: ARRAY[0..cuinMaxConnections] OF T_ADS_ConnectionData;
	
	// Number of ADS (server) connections
	uinNumOfAdsConnections: UINT;
	// Loop variable for request of the handle ID
	uinLoopReqHandle: UINT;
	// Connection index
	uinConIndex: UINT;	
	// Used for generate unique AMS route names
	uinRouteID: UINT;	
END_VAR
VAR CONSTANT
	// Sub states
	cSTA_SUB_INITIALIZE: INT := 500;
	cSTA_SUB_READ: INT := 501;
	cSTA_SUB_READBusy: INT := 502;
	cSTA_SUB_WRITE: INT := 503;
	cSTA_SUB_WRITEBusy: INT := 504;
	cSTA_SUB_RW: INT := 505;
	cSTA_SUB_RWBusy: INT := 506;
	cSTA_SUB_ADD_ROUTE: INT := 507;
	cSTA_SUB_ADD_ROUTEBusy: INT := 508;
	cSTA_SUB_ERROR: INT := 509;
	cSTA_SUB_DONE: INT := 510;
	cSTA_SUB_WAIT_NEXT_POLL: INT := 511;
END_VAR

(*__________________________________________________________________________________________________
¦	
¦	Vistaprint Schweiz GmbH
¦	CH - 8401 Winterthur
¦
¦	www.vistaprint.ch - info@vistaprint.ch
¦___________________________________________________________________________________________________

Function desription:
ADS client for data exchange.
Controls the data exchange between various ADS devices. Devices can be added as server connections to that FUB. 

History:
Version		Date			Author		Comment
---------------------------------------------------------------------------------------------------
0.00.1		05.02.2014		AVME/DSC	Start history
0.00.2		17.02.2014		AVME/DSC	BugZilla 140 - Enter ADS route string automatically during state PONBusy

___________________________________________________________________________________________________*)

IF (me.bolActivate) THEN // cyclic call enabled
	IF (CIf.Info.bolInitDone=FALSE) THEN // first cycle -> init
		CtrlInit();
		CIf.Info.bolInitDone := TRUE;
	ELSE
		CycleStartDuty();
	
		Always();
		
		StateMachine();
		
		CycleEndDuty();
	
	END_IF
END_IF;

METHOD AddConnection
VAR_INPUT
	stConnection: T_ADS_ConnectionData;
END_VAR
// Method adds a connection to the internal list of all ADS connections handled by this block
IF (uinNumOfAdsConnections <= (cuinMaxConnections-1)) THEN
	// Add connection to list
	aListOfConnections[uinNumOfAdsConnections] := stConnection;
	// Assigned connection ID
	aListOfConnections[uinNumOfAdsConnections].udiConID := uinNumOfAdsConnections+1;
	// Inc. number of connections
	uinNumOfAdsConnections:= uinNumOfAdsConnections+1;
END_IF
END_METHOD

METHOD PROTECTED Always : BOOL
SUPER^.Always();

// ----------------------------------------------------------------------------------
// cyclic actions outside of statemachine
IF (me.StateMachine.intState<>cSTA_SINGLE_ANSWER) THEN
	SIf.Cur.uinNumOfAdsConnections:= uinNumOfAdsConnections;	
END_IF

// If no connection added, set alarm and change to state error
IF (uinNumOfAdsConnections = 0) THEN
	// Set Alarm: SIf.Alm[1].strText := 'Initialization error. Minimum one ADS connection must be configured'; 
	pfbAlarmCtrl^.setAlarm(CIf.Info.intCtrlId,1,0,ADR(SIf.Alm),E_AlmState.RST,CIf.Job.eMe_ActivAlmClass);	
	me.StateMachine.intStateNext := BASE_PLC.cSTA_ERROR;
END_IF

// ----------------------------------------------------------------------------------
// Always change actions in Base Library
// ----------------------------------------------------------------------------------
// overrule error always from base -> no EOFF State!! in EOFF go to OFF
IF (me.StateMachine.intStateNext = cSTA_EOFFBusy) THEN
	IF (me.StateMachine.intState=cSTA_OFF) THEN
		me.StateMachine.intStateNext := cSTA_OFF;
	ELSE // stay in OFF
		me.StateMachine.intStateNext := cSTA_OFFBusy;
	END_IF
END_IF
END_METHOD

METHOD FB_init : BOOL
VAR_INPUT
	///if TRUE, the retain variables are initialized (warm start / cold start)
	bInitRetains: BOOL;
	///if TRUE, the instance afterwards gets moved into the copy code (online change)
	bInCopyCode: BOOL;
END_VAR
VAR
	udiTaskCnt: UDINT;
	ii: UINT;
END_VAR
//------------------------------------------------------------------------------------------------------------------------
// to manually change in new FUB implementation!!!
// define valid commands for this controller
FOR ii:= 0 TO (SIZEOF(CIf.Job.aCmdList)/SIZEOF(CIf.Job.aCmdList[0])-1) BY 1 DO
	IF (CIf.Job.aCmdList[ii].intCmd=cCMD_INITIALIZED) THEN
		// found first empty array element
		EXIT;
	END_IF
END_FOR
CIf.Job.aCmdList[ii].intCmd := cCMD_RUN;
CIf.Job.aCmdList[ii].strName := 'Run'; 
CIf.Job.aCmdList[ii].bolAvailable := TRUE;
ii := ii +1;

// set name of class/typ
CIf.Info.strType := 'FB_ACL'; 

// set alarm class
SIf.Alm[1].eAlmClass := E_AlmClass.OFF;
SIf.Alm[1].strText := 'Initialization error. Minimum one ADS connection must be configured'; 
SIf.Alm[2].eAlmClass := E_AlmClass.OFF;
SIf.Alm[2].strText := 'Timeout initialize ADS connection(s)';
SIf.Alm[3].eAlmClass := E_AlmClass.OFF;
SIf.Alm[3].strText := 'Init of ADS connection failed. Note add. info for affected connection ID';
SIf.Alm[4].eAlmClass := E_AlmClass.OFF;
SIf.Alm[4].strText := 'ADS read data failed. Note add. info to get ADS error ID';
SIf.Alm[5].eAlmClass := E_AlmClass.OFF;
SIf.Alm[5].strText := 'ADS write data failed. Note add. info to get ADS error ID';
SIf.Alm[6].eAlmClass := E_AlmClass.OFF;
SIf.Alm[6].strText := 'ADS connection fault. Note add. info for affected connection ID';
SIf.Alm[7].eAlmClass := E_AlmClass.OFF;
SIf.Alm[7].strText :=  'Adding AMS route failed. Note add. info for affected connection ID';

//*******************************************************************************
// initial values
//*******************************************************************************

// software configuration
CIf.SwCfg.bolExist := TRUE;
CIf.SwCfg.bolSimulation := FALSE;

// parameter
SIf.Par.udiTOAddRoute_ms:= 1500;
SIf.Par.udiTOPowerOn_ms:= 10000;
SIf.Par.udiTOReadData_ms:= 1500;
SIf.Par.udiTOWriteData_ms:= 1500;
SIf.Par.udiTORWData_ms:= 1500;
SIf.Par.udiPollingInterval_ms:= 100;
END_METHOD

METHOD PROTECTED getCmdState : STRING
VAR_INPUT
	intCmdState: INT;
	bolState: BOOL;
END_VAR
getCmdState := SUPER^.getCmdState(intCmdState:=intCmdState,bolState:=bolState); // get global/base defined cmds/states
IF (getCmdState='') THEN // global not defined get local
	// get string cmd/state string information in runtime
	IF (bolState=FALSE) THEN
		(*
		// cmd's
		CASE intCmdState OF
			;
		END_CASE
		*)
	ELSE
		// states
		CASE intCmdState OF
			// SUB States
			cSTA_SUB_INITIALIZE:
				getCmdState := 'cSTA_SUB_INITIALIZE';
			cSTA_SUB_READ:
				getCmdState := 'cSTA_SUB_READ';
			cSTA_SUB_READBusy:
				getCmdState := 'cSTA_SUB_READBusy';
			cSTA_SUB_WRITE:
				getCmdState := 'cSTA_SUB_WRITE';
			cSTA_SUB_WRITEBusy:
				getCmdState := 'cSTA_SUB_WRITEBusy';			
			cSTA_SUB_RW:
				getCmdState := 'cSTA_SUB_RW';
			cSTA_SUB_RWBusy:
				getCmdState := 'cSTA_SUB_RWBusy';	
			cSTA_SUB_ADD_ROUTE:
				getCmdState := 'cSTA_SUB_ADD_ROUTE';	
			cSTA_SUB_ADD_ROUTEBusy:
				getCmdState := 'cSTA_SUB_ADD_ROUTEBusy';			
			cSTA_SUB_ERROR:
				getCmdState := 'cSTA_SUB_ERROR';
			cSTA_SUB_DONE:
				getCmdState := 'cSTA_SUB_DONE';
			cSTA_SUB_WAIT_NEXT_POLL:
				getCmdState := 'cSTA_SUB_WAIT_NEXT_POLL';
		END_CASE
	END_IF
END_IF
END_METHOD

METHOD getCtrlSIf : POINTER TO T_Ctrl_SIf_ACL
getCtrlSIf := ADR(SIf);
END_METHOD

METHOD PROTECTED GetNextAccessType : INT
VAR_INPUT
	uinNextConnection:   UINT;
END_VAR
CASE aListOfConnections[uinNextConnection].eAccessType OF	
	E_ADS_AccessType.READ:
		GetNextAccessType:= cSTA_SUB_READ;	
	E_ADS_AccessType.WRITE:
		GetNextAccessType:= cSTA_SUB_WRITE;	
END_CASE
END_METHOD

METHOD NetIDtoAddress: STRING
VAR_INPUT
	strNetID: STRING;
END_VAR
VAR
	intI: INT;
	strCharacter: STRING(1);
	uinExitCounter: UINT;
	cDot: USINT := 16#2E;
END_VAR
// Method convert a ADS NetID to a standard IP Address
// Example: 192.168.70.27.1.1 -> 192.168.70.27
uinExitCounter:=0;
// Get all numbers up to 4 point
FOR intI:=0 TO LEN(strNetID) DO	
	// Get single char
	strCharacter:= Mid(strNetID,1,intI);
	// Incr. exit counter if char = '.'
	IF (F_ToASC(strCharacter) = cDot) THEN
		uinExitCounter:= uinExitCounter +1;
	END_IF
	// As long as 4 point not reached
	IF uinExitCounter < 4 THEN
		NetIDtoAddress:= CONCAT(NetIDtoAddress,strCharacter);	
	ELSE
		EXIT;
	END_IF 
END_FOR
END_METHOD

METHOD PROTECTED sta_ERROR : BOOL
// state implemetation
//--------------------------------------------------------------------------------------
// Entry action
	IF (me.StateMachine.intState<>me.StateMachine.intStateLastCycle) THEN
		me.StateMachine.intStateHistory := me.StateMachine.intStateLastCycle; // -> possibillity to go back to state before error
		me.StateMachine.intStateLastCycle := me.StateMachine.intState;
		
		// Initialize sub state machine
		me.SubStateMachine.intState:= cSTA_SUB_INITIALIZE; 
		me.SubStateMachine.intStateNext := cSTA_SUB_INITIALIZE;
	END_IF

//--------------------------------------------------------------------------------------
// Cyclic action
	IF (me.StateMachine.intState=me.StateMachine.intStateLastCycle) THEN
		// State Change Condition
		IF (CIf.Job.bolAlmReset = TRUE) THEN
			me.StateMachine.intStateNext := cSTA_ERRORQuit;
		END_IF
	END_IF

//--------------------------------------------------------------------------------------
// Exit action
	IF (me.StateMachine.intState<>me.StateMachine.intStateNext) THEN
		;
	END_IF
END_METHOD

METHOD PROTECTED sta_OFF : BOOL
// state implemetation
//--------------------------------------------------------------------------------------
// Entry action
	IF (me.StateMachine.intState<>me.StateMachine.intStateLastCycle) THEN
		me.StateMachine.intStateLastCycle := me.StateMachine.intState;
		// Initialize sub state machine
		me.SubStateMachine.intState:= cSTA_SUB_INITIALIZE; 
		me.SubStateMachine.intStateNext := cSTA_SUB_INITIALIZE;
	END_IF
	
//--------------------------------------------------------------------------------------
// Cyclic action
	IF (me.StateMachine.intState=me.StateMachine.intStateLastCycle) THEN	
		// State Change Condition
		IF (me.Alarm.eActivAlmClass<>E_AlmClass.EOFF) AND (me.Alarm.eActivAlmClass<>E_AlmClass.OFF) THEN	
			IF(me.intCmd=BASE_PLC.cCMD_RUN) THEN
				me.StateMachine.intStateNext := BASE_PLC.cSTA_RUNBusy;
			END_IF
		END_IF
	END_IF

//--------------------------------------------------------------------------------------
// Exit action
	IF (me.StateMachine.intState<>me.StateMachine.intStateNext) THEN
		;
	END_IF
END_METHOD

METHOD PROTECTED sta_PON : BOOL
// state implemetation
//--------------------------------------------------------------------------------------
// Entry action
	IF (me.StateMachine.intState<>me.StateMachine.intStateLastCycle) THEN
		me.StateMachine.intStateLastCycle := me.StateMachine.intState;
		
	END_IF

//--------------------------------------------------------------------------------------
// Cyclic action
	IF (me.StateMachine.intState=me.StateMachine.intStateLastCycle) THEN
		
		;	
		// State Change Condition
		IF (me.intCmd<>cCMD_PON) AND (me.intCmd<>cCMD_DONE) THEN
			me.StateMachine.intStateNext := BASE_PLC.cSTA_OFFBusy;
		END_IF
	END_IF

//--------------------------------------------------------------------------------------
// Exit action
	IF (me.StateMachine.intState<>me.StateMachine.intStateNext) THEN
		;
	END_IF
END_METHOD

METHOD PROTECTED sta_PONBusy : BOOL
VAR
	stRoute: ST_AmsRouteEntry;
	strRouteName: STRING;
END_VAR
// state implemetation
//--------------------------------------------------------------------------------------
// Entry action
	IF (me.StateMachine.intState<>me.StateMachine.intStateLastCycle) THEN
		me.StateMachine.intStateLastCycle := me.StateMachine.intState;
		
		uinRouteID:= 0;
		uinConIndex:=0;
		// Initialize sub state machine
		me.SubStateMachine.intState:= cSTA_SUB_ADD_ROUTE; 
		me.SubStateMachine.intStateNext := cSTA_SUB_ADD_ROUTE;
		
	END_IF

//--------------------------------------------------------------------------------------
// Cyclic action
	IF (me.StateMachine.intState=me.StateMachine.intStateLastCycle) THEN
		
			// Sub statemachine to set necessary AMS routes and determine the handle ID of all connections in list	
			CASE me.SubStateMachine.intState OF	
			
				// **************************************************************************
				// Call fbAddRoute to add AMS route. Block automatically check if NetID or Name already exist.
				// Double entries not possible!
				// **************************************************************************
				cSTA_SUB_ADD_ROUTE:
				
					// Prepare unique AMS route name: Controller Name: + ID
					uinRouteID:= uinRouteID + 1;
					strRouteName := CONCAT(CIf.Info.strName, ': ID');
					strRouteName := CONCAT(strRouteName, UINT_TO_STRING(uinRouteID));
							
					// Prepare route data
					stRoute.sName:= strRouteName;
					stRoute.sNetID:= aListOfConnections[uinConIndex].strNetID;
					stRoute.sAddress:= THIS^.NetIDtoAddress(aListOfConnections[uinConIndex].strNetID);
					stRoute.eTransport:= eRouteTransport_TCP_IP;
				
					// Add route
					fbAddRoute(bExecute	:= FALSE);
					fbAddRoute( sNetID 	:= '',
								stRoute	:= stRoute,
								bExecute:= TRUE,
								tTimeout:= UDINT_TO_TIME(SIf.Par.udiTOAddRoute_ms),
								bBusy	=>,
								bError	=>,
								nErrID	=>);
				
					me.SubStateMachine.intStateNext := cSTA_SUB_ADD_ROUTEBusy;		
							
				// **************************************************************************
				// Add route busy
				// **************************************************************************
				cSTA_SUB_ADD_ROUTEBusy:
				
					fbAddRoute(bExecute:= FALSE);
					// Add route done
					IF NOT (fbAddRoute.bBusy) THEN
						IF NOT (fbAddRoute.bError) THEN
							// More connections?
							IF (uinConIndex < (uinNumOfAdsConnections-1)) THEN
								uinConIndex:= uinConIndex+1;
								me.SubStateMachine.intStateNext := cSTA_SUB_ADD_ROUTE;
							// All routes added - go on with determine the handle ID 
							ELSE
								uinConIndex:=0;
								me.SubStateMachine.intStateNext := cSTA_SUB_RW;	
							END_IF
						// Error
						ELSE
							// SIf.Alm[7].strText :=  'Adding AMS route failed. Note add. info for affected connection ID';
							pfbAlarmCtrl^.setAlarm(CIf.Info.intCtrlId,7,UDINT_TO_DINT(aListOfConnections[uinConIndex].udiConID),ADR(SIf.Alm),E_AlmState.RST,CIf.Job.eMe_ActivAlmClass);
							me.SubStateMachine.intStateNext := cSTA_SUB_ERROR;		
						END_IF
					END_IF
			
				// **************************************************************************
				// Call fbReadWrite to determine the handle ID
				// **************************************************************************
				cSTA_SUB_RW:
			
					fbReadWrite(WRTRD:= FALSE);
    				fbReadWrite(NETID		:= aListOfConnections[uinConIndex].strNetID,
                				PORT		:= aListOfConnections[uinConIndex].uinTargetPort,
                   				IDXGRP		:= cGET_SYMHANDLE_BYNAME,  
                   				IDXOFFS     := 16#0000,
                   				WRITELEN    := INT_TO_UDINT(LEN(aListOfConnections[uinConIndex].strRoute)+1),
								READLEN     := SIZEOF(aListOfConnections[uinConIndex].udiHandle),
								SRCADDR     := ADR(aListOfConnections[uinConIndex].strRoute),
								DESTADDR    := ADR(aListOfConnections[uinConIndex].udiHandle),
								WRTRD       := TRUE,
								TMOUT       := UDINT_TO_TIME(SIf.Par.udiTORWData_ms),
								BUSY        => ,
								ERR         => ,
								ERRID       => );
								
					me.SubStateMachine.intStateNext := cSTA_SUB_RWBusy;		
				
				// **************************************************************************
				// Read/Write busy
				// **************************************************************************
				cSTA_SUB_RWBusy:
					fbReadWrite(WRTRD:= FALSE);
					// Read/Write done
					IF NOT (fbReadWrite.BUSY) THEN
						IF NOT (fbReadWrite.ERR) THEN
							// More connections?
							IF (uinConIndex < (uinNumOfAdsConnections-1)) THEN
								uinConIndex:= uinConIndex+1;
								me.SubStateMachine.intStateNext := cSTA_SUB_RW;
							// Done - all connection handles are determined 
							ELSE
								me.SubStateMachine.intStateNext := cSTA_SUB_DONE;	
							END_IF
						// Error
						ELSE
							// SIf.Alm[3].strText := 'Init of ADS connection failed. Check add. info for affected connection ID';
							pfbAlarmCtrl^.setAlarm(CIf.Info.intCtrlId,3,UDINT_TO_DINT(aListOfConnections[uinConIndex].udiConID),ADR(SIf.Alm),E_AlmState.RST,CIf.Job.eMe_ActivAlmClass);
							me.SubStateMachine.intStateNext := cSTA_SUB_ERROR;		
						END_IF
					END_IF
				
				// **************************************************************************
				// All necessary AMS routes set and connection handles are determined 
				// **************************************************************************
				cSTA_SUB_DONE:
				
				// **************************************************************************
				// Error
				// **************************************************************************
				cSTA_SUB_ERROR:
				
			END_CASE	
			
		
		// State Change Condition
		IF ((me.SubStateMachine.intState=cSTA_SUB_ERROR) OR (me.StateMachine.udiTimeInState_ms >= SIf.Par.udiTOPowerOn_ms)) THEN
			// In case if TO
			IF (me.StateMachine.udiTimeInState_ms >= SIf.Par.udiTOPowerOn_ms) THEN
				// SIf.Alm[2].strText := 'Timeout initialize ADS connection(s)';
				pfbAlarmCtrl^.setAlarm(CIf.Info.intCtrlId,2,UDINT_TO_DINT(me.StateMachine.udiTimeInState_ms),ADR(SIf.Alm),E_AlmState.RST,CIf.Job.eMe_ActivAlmClass);
			END_IF
			me.StateMachine.intStateNext := cSTA_ERROR;				
		ELSIF (me.SubStateMachine.intState=cSTA_SUB_DONE) THEN
			me.StateMachine.intStateNext := cSTA_PON;
		END_IF
			
	END_IF

//--------------------------------------------------------------------------------------
// Exit action
	IF (me.StateMachine.intState<>me.StateMachine.intStateNext) THEN
		;
	END_IF
END_METHOD

METHOD PROTECTED sta_RUN : BOOL
// state implemetation
//--------------------------------------------------------------------------------------
// Entry action
	IF (me.StateMachine.intState<>me.StateMachine.intStateLastCycle) THEN
		me.StateMachine.intStateLastCycle := me.StateMachine.intState;
					
		uinConIndex:=0;
		// Initialize sub state machine
		me.SubStateMachine.intState:= cSTA_SUB_INITIALIZE; 
		me.SubStateMachine.intStateNext := cSTA_SUB_INITIALIZE;
	END_IF

//--------------------------------------------------------------------------------------
// Cyclic action
	IF (me.StateMachine.intState=me.StateMachine.intStateLastCycle) THEN

		// Sub statemachine to handle all connections in list dependent access type (read, write, rw)
		CASE me.SubStateMachine.intState OF	
	
			//************************************************************************
			// Initialize
			//************************************************************************
			cSTA_SUB_INITIALIZE:
				// Get access type
				me.SubStateMachine.intStateNext:= THIS^.GetNextAccessType(uinConIndex);
							
			//************************************************************************					
			// Call fbRead
			//************************************************************************
			cSTA_SUB_READ:
		
				fbRead(READ:= FALSE);
				fbRead(NETID       := aListOfConnections[uinConIndex].strNetID,
						PORT       := aListOfConnections[uinConIndex].uinTargetPort,
						IDXGRP     := cREAD_WRITE_SYMVAL_BYHANDLE,
						IDXOFFS    := aListOfConnections[uinConIndex].udiHandle,
						LEN        := aListOfConnections[uinConIndex].udiDataLen,
						DESTADDR   := aListOfConnections[uinConIndex].pData,
						READ       := TRUE,
						TMOUT      := UDINT_TO_TIME(SIf.Par.udiTOReadData_ms),
						BUSY       => ,
						ERR        => ,
						ERRID      => );
														
				me.SubStateMachine.intStateNext := cSTA_SUB_READBusy;			
							
			//************************************************************************
			// Read busy
			//************************************************************************
			cSTA_SUB_READBusy:
				fbRead(READ:= FALSE);
				// Read done
				IF NOT (fbRead.BUSY) THEN
					IF NOT (fbRead.ERR) THEN	
						// More connections?
						IF (uinConIndex < (uinNumOfAdsConnections-1)) THEN
							uinConIndex:= uinConIndex+1;
							// Get next access type
							me.SubStateMachine.intStateNext:= THIS^.GetNextAccessType(uinConIndex);
						// Done - all connection handles are determined 
						ELSE
							me.SubStateMachine.intStateNext := cSTA_SUB_WAIT_NEXT_POLL;	
						END_IF						
					// Error
					ELSE
						// SIf.Alm[4].strText := 'ADS read data failed. Note add. info to get ADS error ID';
						pfbAlarmCtrl^.setAlarm(CIf.Info.intCtrlId,4,UDINT_TO_DINT(fbRead.ERRID),ADR(SIf.Alm),E_AlmState.RST,CIf.Job.eMe_ActivAlmClass);
						me.SubStateMachine.intStateNext := cSTA_SUB_ERROR;		
					END_IF
				END_IF	
				
			//************************************************************************					
			// Call fbWrite
			//************************************************************************
			cSTA_SUB_WRITE:
		
				fbWrite(WRITE:= FALSE);
				fbWrite(NETID      := aListOfConnections[uinConIndex].strNetID,
						PORT       := aListOfConnections[uinConIndex].uinTargetPort,
						IDXGRP     := cREAD_WRITE_SYMVAL_BYHANDLE,
						IDXOFFS    := aListOfConnections[uinConIndex].udiHandle,
						LEN        := aListOfConnections[uinConIndex].udiDataLen,
						SRCADDR    := aListOfConnections[uinConIndex].pData,
						WRITE      := TRUE,
						TMOUT      := UDINT_TO_TIME(SIf.Par.udiTOWriteData_ms),
						BUSY       => ,
						ERR        => ,
						ERRID      => );
														
				me.SubStateMachine.intStateNext := cSTA_SUB_WRITEBusy;		
				
			//************************************************************************
			// Write busy
			//************************************************************************
			cSTA_SUB_WRITEBusy:
				fbWrite(WRITE:= FALSE);
				// Write done
				IF NOT (fbWrite.BUSY) THEN
					IF NOT (fbWrite.ERR) THEN
						// More connections?
						IF (uinConIndex < (uinNumOfAdsConnections-1)) THEN
							uinConIndex:= uinConIndex+1;
							// Get next access type
							me.SubStateMachine.intStateNext:= THIS^.GetNextAccessType(uinConIndex);
						// Done - all connection handles are determined 
						ELSE
							me.SubStateMachine.intStateNext := cSTA_SUB_WAIT_NEXT_POLL;	
						END_IF
					// Error
					ELSE
						// SIf.Alm[5].strText := 'ADS write data failed. Note add. info to get ADS error ID';
						pfbAlarmCtrl^.setAlarm(CIf.Info.intCtrlId,5,UDINT_TO_DINT(fbWrite.ERRID),ADR(SIf.Alm),E_AlmState.RST,CIf.Job.eMe_ActivAlmClass);
						me.SubStateMachine.intStateNext := cSTA_SUB_ERROR;		
					END_IF
				END_IF			
		
			//************************************************************************
			// Wait for next polling - Connection list completely processed 
			//************************************************************************	
			cSTA_SUB_WAIT_NEXT_POLL:
			
				// Wait polling time expired 	
				IF (me.SubStateMachine.udiTimeInState_ms >= SIf.Par.udiPollingInterval_ms) THEN				
					//Start again at first connection in list
					uinConIndex:=0;
					me.SubStateMachine.intStateNext := cSTA_SUB_INITIALIZE;
				END_IF
				
			//************************************************************************
			// ERROR			
			//************************************************************************	
			cSTA_SUB_ERROR:
				// SIf.Alm[6].strText := 'ADS connection fault. Note add. info for affected connection ID';
				pfbAlarmCtrl^.setAlarm(CIf.Info.intCtrlId,6,UDINT_TO_DINT(aListOfConnections[uinConIndex].udiConID),ADR(SIf.Alm),E_AlmState.RST,CIf.Job.eMe_ActivAlmClass);
				me.StateMachine.intStateNext := BASE_PLC.cSTA_ERROR;	
			
		END_CASE			
	END_IF

//--------------------------------------------------------------------------------------
// Exit action
	IF (me.StateMachine.intState<>me.StateMachine.intStateNext) THEN
		;
	END_IF
END_METHOD

METHOD PROTECTED sta_RUNBusy : BOOL
// state implemetation
//--------------------------------------------------------------------------------------
// Entry action
	IF (me.StateMachine.intState<>me.StateMachine.intStateLastCycle) THEN
		me.StateMachine.intStateLastCycle := me.StateMachine.intState;
		;
	END_IF

//--------------------------------------------------------------------------------------
// Cyclic action
	IF (me.StateMachine.intState=me.StateMachine.intStateLastCycle) THEN
		IF (TRUE) THEN
			me.StateMachine.intStateNext := BASE_PLC.cSTA_RUN;
		END_IF
	END_IF

//--------------------------------------------------------------------------------------
// Exit action
	IF (me.StateMachine.intState<>me.StateMachine.intStateNext) THEN
		;
	END_IF
END_METHOD

METHOD PROTECTED StateMachine : BOOL
SUPER^.StateMachine();

// main statemachine of base controller
CASE me.StateMachine.intState OF
	cSTA_RUNBusy: 
        THIS^.sta_RUNBusy();
    cSTA_RUN: 
        THIS^.sta_RUN();				
END_CASE;
END_METHOD

END_FUNCTION_BLOCK

// POUs/Controller/Driver/BCD (Bar code driver)/FB_BCD
FUNCTION_BLOCK FB_BCD
VAR
	bolInitDone: BOOL;
	bolActivate: BOOL := TRUE;
	/// driver specific interface
	SIf: T_BCD;
	stStateMachine: T_BCD_StateMachine;
	stSubStateMachine: T_BCD_StateMachine;
	/// Create/release TCP/IP connection
	fbClientConnection: FB_ClientServerConnection;
	/// Send TCP/IP data
	fbSend: FB_SocketSend;
	/// Receive TCP/IP data
	fbReceive: FB_SocketReceive;
	/// Rx data buffer
	aRxData: ARRAY[0..300] OF BYTE;
	/// Tx data buffer
	aTxData: ARRAY[0..300] OF BYTE;
	intTxState: INT;
	bolExecuteSend: BOOL;
	/// counter for sended frames 
	udiNSend: UDINT;
	intRxState: INT;
	bolExecuteRead: BOOL;
	/// Count of received data bytes
	udiReceivedBytes: UDINT;
	strReceivedMessage: STRING(255);
END_VAR
VAR CONSTANT
	cBCD_SUB_Send: INT := 2000;
	cBCD_SUB_Wait: INT := 2001;
	cBCD_SUB_Read: INT := 2002;
	cBCD_SUB_CheckAnswer: INT := 2003;
	cBCD_SUB_GetData: INT := 2004;
	cBCD_SUB_Done: INT := 2005;
	cBCD_SUB_Error: INT := 2006;
	cTxIdle: USINT := 0;
	cTxBusy: USINT := 1;
	cRxIdle: USINT := 0;
	cRxBusy: USINT := 1;
	cRxConv: USINT := 2;
	cSTX: USINT := 16#2;
	cETX: USINT := 16#3;
	cCR: USINT := 16#D;
	cLF: USINT := 16#A;
END_VAR

(*__________________________________________________________________________________________________
¦	
¦	Vistaprint Schweiz GmbH
¦	CH - 8401 Winterthur
¦
¦	www.vistaprint.ch - info@vistaprint.ch
¦___________________________________________________________________________________________________

Function desription:
TCP-IP driver for SICK barcode reader CLV632-0120
Note: This driver work as a TCP client.

History:
Version		Date			Author		Comment
---------------------------------------------------------------------------------------------------
0.00.1		18.12.2013		AVME/DSC	Start history
0.00.2		03.01.2014		AVME/DSC	Basic functionalities implemented and tested. Following commands are supported:
										CMD_CONNECT_SOCKET 	1002 		// Connect TCP socket
										CMD_CLOSE_SOCKET 	1004 		// Close TCP socket
										CMD_COM_TEST 		1006 		// Communication test 
										CMD_READ_BARCODE 	1014 		// Command enable the sensor gate for X-TIME ("duration" setting of sensor object trigger)
																		// Sensor try to detect a barcode.
0.00.3		27.01.2014		AVME/DSC    Added new method "CheckSensorError" to set "bolSensorError" in case if sensor answer with SOPAS error																					 							
		
___________________________________________________________________________________________________*)


IF (bolActivate) THEN // cyclic call enabled
	
	IF (bolInitDone=FALSE) THEN // first cycle -> init
		CtrlInit();	
		bolInitDone := TRUE;
	ELSE
		CycleStartDuty();
				
		StateMachine();
		
		CycleEndDuty();
	END_IF
	
END_IF;

METHOD PRIVATE CheckSensorError
VAR
	strErrorID: STRING(3);
	bytErrorID: BYTE;
	cbData: UDINT;
END_VAR
(*--------------------------------------------------------------------------
IF an error occurs the Sopas command is answered with:
[STX]sFA <x>[ETX] as an error response

	Error list: <x> can have following values:
	1:	Access denied
	2:	Unknown Index
	3:	Unknown Index
	4:	Wrong Condition
	5:	Invalid Data
	6:	Unknown Error
	7:	Too Many Parameter
	8:	Parameter Missing
	9: 	Wrong Parameter
	A:	No Write Access
	B:	Unknown Command
	C:	Unknown Command
	D:	Server Busy
	E:	Textstring Too Long
	F:	Unknown Event
	10:	Too many Parameter
	11: Invalid Character
	12.	No Message
	13:	No Answer
	14:	Internal Error
	15:	HubAddress: wrong
	16:	HubAddress: error
	17:	HubAddress: error

---------------------------------------------------------------------------*)

// If received message is an error response from sensor: [STX]sFA <x>[ETX]    				
IF (TC2_STANDARD.FIND(strReceivedMessage,'sFA') <> 0) THEN
	
	// Get error number
	strErrorID := Mid(strReceivedMessage,LEN(strReceivedMessage)-1,5);
	cbData := HEXSTR_TO_DATA( strErrorID, ADR(bytErrorID), SIZEOF(bytErrorID));

	// No interpretation of the error number, only set SensorError with error number info 
	(*
	CASE bytErrorID OF
		16#1: 
		16#2:
		16#3:	
		16#A:			
		16#B,16#C:
	END_CASE
	*)
	
	IF (SIf.stErr.bolErrorActive = FALSE) THEN
		SIf.stErr.bolErrorActive:= TRUE;	
		SIf.stErr.bolSensorError:= TRUE; 
		SIf.stErr.udiErrorID := bytErrorID;	
		// Try to close the socket. Needs reconnect for socket after an error!	
		stStateMachine.intStateNext := cBCD_STA_CloseSocketBusy;	
	END_IF	

END_IF
END_METHOD

METHOD PROTECTED CtrlInit : BOOL
// one time first cyclic call
// The socket is closed
stStateMachine.intStateNext := cBCD_STA_SocketClosed;
END_METHOD

METHOD PROTECTED CycleEndDuty : BOOL
SIf.strState := THIS^.getCmdState(intCmdState:=stStateMachine.intState,bolState:=TRUE);

IF (stStateMachine.intState<>stStateMachine.intStateNext) THEN
	stStateMachine.intState := stStateMachine.intStateNext;  // set next state for next cycle
END_IF

(***************************************************************
        Function Block Calls
***************************************************************)

// Cyclic call of method "HandleTxData"
THIS^.HandleTxData();
END_METHOD

METHOD PROTECTED CycleStartDuty : BOOL
// ----------------------------------------------------------------------------------
// cyclic actions outside of statemachine

// Simulation active
IF (SIf.stCfg.bolSimulation) THEN
	;
ELSE
	;
END_IF

// Cyclic call of the client connection
fbClientConnection();
// Cyclic call of method "HandleRxData"
THIS^.HandleRxData();

